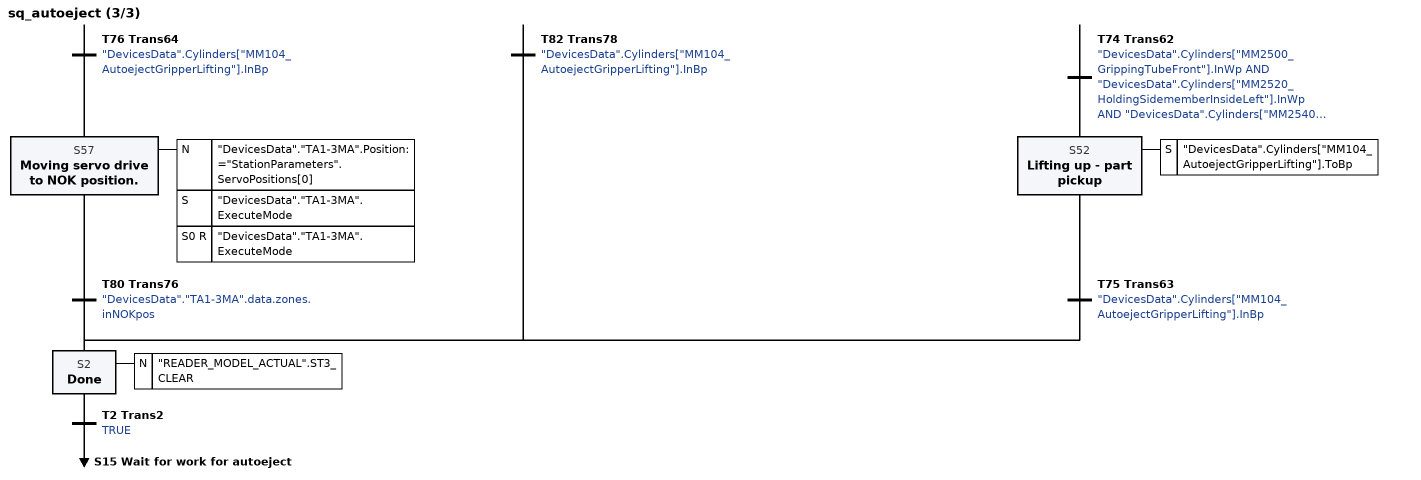
   // sequencer 1
   INITIAL_STEP Init:   // S1, max time T#10S, warning time T#7S
   END_STEP
   TRANSITION Trans1 FROM Init TO "Checking gripper status"   // T1
      := ("ModeSelection_DB".mode.activeMode = "mode_2_base") OR (("ModeSelection_DB".mode.activeMode = "mode_4_semiautomat") AND #start);
   END_TRANSITION
   STEP Done:   // S2, max time T#10S, warning time T#7S
              N    "READER_MODEL_ACTUAL".ST3_CLEAR
   END_STEP
   TRANSITION Trans2 FROM Done TO "Wait for work for autoeject"   // T2, jump
      := TRUE;
   END_TRANSITION
   STEP "Base done":   // S12, max time T#10S, warning time T#7S
   END_STEP
   TRANSITION Trans17 FROM "Base done" TO "Wait for work for autoeject"   // T17
      := (("ModeSelection_DB".mode.activeMode = "mode_3_automat") OR (("ModeSelection_DB".mode.activeMode = "mode_4_semiautomat") AND #start)) AND (#"Base done".T > t#2000MS);
   END_TRANSITION
   STEP "Wait for work for autoeject":   // S15, max time T#10S, warning time T#7S
   END_STEP
   TRANSITION "OK dropoff" FROM "Wait for work for autoeject" TO "Moving servo drive to OK position"   // T22
      := (("ModeSelection_DB".mode.activeMode = "mode_3_automat") OR (("ModeSelection_DB".mode.activeMode = "mode_4_semiautomat") AND #start)) AND "iR1outOf_AE_left_bottom" AND "iR1outOf_AE_left_top" AND "iR1outOf_AE_right_bottom" AND "iR1outOf_AE_right_top" AND "AutoPositions".AE_Gripper.PartPresent AND "AutoPositions".AE_Gripper.StFinished[3] AND NOT "AutoPositions".AE_Gripper.PartNOK AND "iAEtubePresentFront" AND "iAEtubePresentRear" AND NOT "AutoPositions".St4_OKposition.PartPresent AND NOT "i4partPresent";
   END_TRANSITION
   TRANSITION "NOK dropoff" FROM "Wait for work for autoeject" TO "Moving servo drive to NOK position.."   // T23
      := (("ModeSelection_DB".mode.activeMode = "mode_3_automat") OR (("ModeSelection_DB".mode.activeMode = "mode_4_semiautomat") AND #start)) AND "iR1outOf_AE_left_bottom" AND "iR1outOf_AE_left_top" AND "iR1outOf_AE_right_bottom" AND "iR1outOf_AE_right_top" AND "AutoPositions".AE_Gripper.PartPresent AND (NOT "AutoPositions".AE_Gripper.StFinished[3] OR "AutoPositions".AE_Gripper.PartNOK) AND "iAEtubePresentFront" AND "iAEtubePresentRear" AND NOT "PartHolderData".NOKBoxFull;
   END_TRANSITION
   TRANSITION "jig pickup" FROM "Wait for work for autoeject" TO "Moving servo drive to jig (st3) position"   // T21
      := (("ModeSelection_DB".mode.activeMode = "mode_3_automat") OR (("ModeSelection_DB".mode.activeMode = "mode_4_semiautomat") AND #start)) AND "iR1outOf_AE_left_bottom" AND "iR1outOf_AE_left_top" AND "iR1outOf_AE_right_bottom" AND "iR1outOf_AE_right_top" AND "AutoPositions".St3_Fitting.PartPresent AND "i3partPresent" AND NOT "AutoPositions".AE_Gripper.PartPresent AND NOT "iAEtubePresentFront" AND NOT "iAEtubePresentRear" AND NOT "AutoPositions".St4_OKposition.PartPresent AND NOT "i4partPresent";
   END_TRANSITION
   STEP "Close gripper - part pickup":   // S51, max time T#10S, warning time T#7S
              S    "DevicesData".Cylinders["MM2500_GrippingTubeFront"].ToWp
              S    "DevicesData".Cylinders["MM2520_HoldingSidememberInsideLeft"].ToWp
              S    "DevicesData".Cylinders["MM2540_HoldingSidememberOutsideLeft"].ToWp
   END_STEP
   TRANSITION Trans62 FROM "Close gripper - part pickup" TO "Lifting up - part pickup"   // T74
      := "DevicesData".Cylinders["MM2500_GrippingTubeFront"].InWp AND "DevicesData".Cylinders["MM2520_HoldingSidememberInsideLeft"].InWp AND "DevicesData".Cylinders["MM2540_HoldingSidememberOutsideLeft"].InWp;
   END_TRANSITION
   STEP "Open gripper - OK part dropoff":   // S53, max time T#10S, warning time T#7S
              S    "DevicesData".Cylinders["MM2500_GrippingTubeFront"].ToBp
              S    "DevicesData".Cylinders["MM2520_HoldingSidememberInsideLeft"].ToBp
              S    "DevicesData".Cylinders["MM2540_HoldingSidememberOutsideLeft"].ToBp
   END_STEP
   TRANSITION Trans75 FROM "Open gripper - OK part dropoff" TO "Lifting up - OK part dropoff"   // T79
      := "DevicesData".Cylinders["MM2500_GrippingTubeFront"].InBp AND "DevicesData".Cylinders["MM2520_HoldingSidememberInsideLeft"].InBp AND "DevicesData".Cylinders["MM2540_HoldingSidememberOutsideLeft"].InBp;
   END_TRANSITION
   STEP "Moving servo drive to OK position":   // S54, max time T#30S, warning time T#7S
      supervision V := #"Moving servo drive to OK position".T > #"Moving servo drive to OK position".T_MAX;
              N    "DevicesData"."TA1-3MA".Position:="StationParameters".ServoPositions[1]
              S    "DevicesData"."TA1-3MA".ExecuteMode
          S0  R    "DevicesData"."TA1-3MA".ExecuteMode
   END_STEP
   TRANSITION Trans74 FROM "Moving servo drive to OK position" TO "Lifting down - OK part dropoff"   // T78
      := "DevicesData"."TA1-3MA".data.zones.inOKpos;
   END_TRANSITION
   STEP "Lifting up - OK part dropoff":   // S55, max time T#10S, warning time T#7S
              S    "DevicesData".Cylinders["MM104_AutoejectGripperLifting"].ToBp
   END_STEP
   TRANSITION Trans64 FROM "Lifting up - OK part dropoff" TO "Moving servo drive to NOK position."   // T76
      := "DevicesData".Cylinders["MM104_AutoejectGripperLifting"].InBp;
   END_TRANSITION
   STEP "Lifting down - OK part dropoff":   // S56, max time T#10S, warning time T#7S
              S    "DevicesData".Cylinders["MM104_AutoejectGripperLifting"].ToWp
   END_STEP
   TRANSITION Trans73 FROM "Lifting down - OK part dropoff" TO "Open gripper - OK part dropoff"   // T77
      := "DevicesData".Cylinders["MM104_AutoejectGripperLifting"].InWp;
   END_TRANSITION
   STEP "Moving servo drive to jig (st3) position":   // S49, max time T#30S, warning time T#7S
      supervision V := #"Moving servo drive to jig (st3) position".T > #"Moving servo drive to jig (st3) position".T_MAX;
              N    "DevicesData"."TA1-3MA".Position:="StationParameters".ServoPositions[2]
              S    "DevicesData"."TA1-3MA".ExecuteMode
          S0  R    "DevicesData"."TA1-3MA".ExecuteMode
   END_STEP
   TRANSITION Trans85 FROM "Moving servo drive to jig (st3) position" TO "Waiting for part to be finished"   // T85
      := "DevicesData"."TA1-3MA".data.zones.inST3jig;
   END_TRANSITION
   STEP "Lifting up - part pickup":   // S52, max time T#10S, warning time T#7S
              S    "DevicesData".Cylinders["MM104_AutoejectGripperLifting"].ToBp
   END_STEP
   TRANSITION Trans63 FROM "Lifting up - part pickup" TO Done   // T75
      := "DevicesData".Cylinders["MM104_AutoejectGripperLifting"].InBp;
   END_TRANSITION
   STEP "Lifting down - part pickup":   // S50, max time T#10S, warning time T#7S
              S    "DevicesData".Cylinders["MM104_AutoejectGripperLifting"].ToWp
   END_STEP
   TRANSITION Trans61 FROM "Lifting down - part pickup" TO "Close gripper - part pickup"   // T73
      := "DevicesData".Cylinders["MM104_AutoejectGripperLifting"].InWp;
   END_TRANSITION
   STEP "Checking gripper status":   // S37, max time T#10S, warning time T#7S
   END_STEP
   TRANSITION "base w/o part" FROM "Checking gripper status" TO "Open gripper"   // T56
      := NOT "AutoPositions".AE_Gripper.PartPresent AND NOT "iAEtubePresentFront" AND NOT "iAEtubePresentRear";
   END_TRANSITION
   TRANSITION "base w/ part" FROM "Checking gripper status" TO "Close gripper"   // T57
      := "AutoPositions".AE_Gripper.PartPresent AND "iAEtubePresentFront" AND "iAEtubePresentRear";
   END_TRANSITION
   STEP "Open gripper":   // S38, max time T#10S, warning time T#7S
              S    "DevicesData".Cylinders["MM2500_GrippingTubeFront"].ToBp
              S    "DevicesData".Cylinders["MM2520_HoldingSidememberInsideLeft"].ToBp
              S    "DevicesData".Cylinders["MM2540_HoldingSidememberOutsideLeft"].ToBp
   END_STEP
   TRANSITION Trans58 FROM "Open gripper" TO "Lifting up"   // T58
      := "DevicesData".Cylinders["MM2500_GrippingTubeFront"].InBp AND "DevicesData".Cylinders["MM2520_HoldingSidememberInsideLeft"].InBp AND "DevicesData".Cylinders["MM2540_HoldingSidememberOutsideLeft"].InBp;
   END_TRANSITION
   STEP "Close gripper":   // S39, max time T#10S, warning time T#7S
              S    "DevicesData".Cylinders["MM2500_GrippingTubeFront"].ToWp
              S    "DevicesData".Cylinders["MM2520_HoldingSidememberInsideLeft"].ToWp
              S    "DevicesData".Cylinders["MM2540_HoldingSidememberOutsideLeft"].ToWp
   END_STEP
   TRANSITION Trans59 FROM "Close gripper" TO "Lifting up"   // T59
      := "DevicesData".Cylinders["MM2500_GrippingTubeFront"].InWp AND "DevicesData".Cylinders["MM2520_HoldingSidememberInsideLeft"].InWp AND "DevicesData".Cylinders["MM2540_HoldingSidememberOutsideLeft"].InWp;
   END_TRANSITION
   STEP "Lifting up":   // S40, max time T#10S, warning time T#7S
              S    "DevicesData".Cylinders["MM104_AutoejectGripperLifting"].ToBp
   END_STEP
   TRANSITION Trans60 FROM "Lifting up" TO "Checking homing status"   // T60
      := "DevicesData".Cylinders["MM104_AutoejectGripperLifting"].InBp;
   END_TRANSITION
   STEP "Checking homing status":   // S41, max time T#10S, warning time T#7S
   END_STEP
   TRANSITION referenced FROM "Checking homing status" TO "Checking robot position."   // T61
      := "DevicesData"."TA1-3MA".AxisRef;
   END_TRANSITION
   TRANSITION "not refrenced" FROM "Checking homing status" TO "Checking robot position"   // T62
      := NOT "DevicesData"."TA1-3MA".AxisRef;
   END_TRANSITION
   STEP "Checking robot position":   // S42, max time T#10S, warning time T#7S
   END_STEP
   TRANSITION "out of zones" FROM "Checking robot position" TO "Switch servo to homing mode"   // T63
      := "iR1outOf_AE_left_bottom" AND "iR1outOf_AE_left_top" AND "iR1outOf_AE_right_bottom" AND "iR1outOf_AE_right_top";
   END_TRANSITION
   TRANSITION "in zones" FROM "Checking robot position" TO "You have to move robot out of the autoeject zones manually"   // T64
      := TRUE;
   END_TRANSITION
   STEP "Switch servo to homing mode":   // S43, max time T#10S, warning time T#7S
      supervision V := #"Switch servo to homing mode".T > #"Switch servo to homing mode".T_MAX;
              N    "DevicesData"."TA1-3MA".ModePos:=4
   END_STEP
   TRANSITION Trans65 FROM "Switch servo to homing mode" TO "Homing servo drive"   // T65
      := "DevicesData"."TA1-3MA".ActMode = 4;
   END_TRANSITION
   STEP "You have to move robot out of the autoeject zones manually":   // S44, max time T#10S, warning time T#7S
      supervision V := "AlwaysTRUE";
   END_STEP
   TRANSITION Trans66 FROM "You have to move robot out of the autoeject zones manually" TO END   // T66
      := NOT "AlwaysTRUE";
   END_TRANSITION
   STEP "Homing servo drive":   // S45, max time T#30S, warning time T#7S
      supervision V := #"Homing servo drive".T > #"Homing servo drive".T_MAX;
              S    "DevicesData"."TA1-3MA".ExecuteMode
          S0  R    "DevicesData"."TA1-3MA".ExecuteMode
   END_STEP
   TRANSITION Trans67 FROM "Homing servo drive" TO "Checking robot position."   // T67
      := "DevicesData"."TA1-3MA".AxisRef AND "DevicesData"."TA1-3MA".AxisPosOk;
   END_TRANSITION
   STEP "Checking robot position.":   // S46, max time T#10S, warning time T#7S
   END_STEP
   TRANSITION Trans68 FROM "Checking robot position." TO "Switch servo to positioning mode"   // T68
      := ("iR1outOf_AE_left_bottom" AND "iR1outOf_AE_left_top" AND "iR1outOf_AE_right_bottom" AND "iR1outOf_AE_right_top") OR ("iR1outOf_AE_right_bottom" AND "iR1outOf_AE_right_top" AND "DevicesData"."TA1-3MA".data.zones.outOfST3zone);
   END_TRANSITION
   TRANSITION Trans69 FROM "Checking robot position." TO "You have to move robot out of the autoeject zones manually"   // T69, jump
      := TRUE;
   END_TRANSITION
   STEP "Switch servo to positioning mode":   // S47, max time T#10S, warning time T#7S
      supervision V := #"Switch servo to positioning mode".T > #"Switch servo to positioning mode".T_MAX;
              N    "DevicesData"."TA1-3MA".ModePos:=2
   END_STEP
   TRANSITION Trans70 FROM "Switch servo to positioning mode" TO Timeout   // T70
      := "DevicesData"."TA1-3MA".ActMode = 2;
   END_TRANSITION
   STEP "Moving servo drive to NOK position":   // S48, max time T#30S, warning time T#7S
      supervision V := #"Moving servo drive to NOK position".T > #"Moving servo drive to NOK position".T_MAX;
              N    "DevicesData"."TA1-3MA".Position:="StationParameters".ServoPositions[0]
              S    "DevicesData"."TA1-3MA".ExecuteMode
          S0  R    "DevicesData"."TA1-3MA".ExecuteMode
   END_STEP
   TRANSITION Trans71 FROM "Moving servo drive to NOK position" TO "Base done"   // T71
      := "DevicesData"."TA1-3MA".data.zones.inNOKpos;
   END_TRANSITION
   STEP "Moving servo drive to NOK position.":   // S57, max time T#30S, warning time T#7S
      supervision V := #"Moving servo drive to NOK position.".T > #"Moving servo drive to NOK position.".T_MAX;
              N    "DevicesData"."TA1-3MA".Position:="StationParameters".ServoPositions[0]
              S    "DevicesData"."TA1-3MA".ExecuteMode
          S0  R    "DevicesData"."TA1-3MA".ExecuteMode
   END_STEP
   TRANSITION Trans76 FROM "Moving servo drive to NOK position." TO Done   // T80
      := "DevicesData"."TA1-3MA".data.zones.inNOKpos;
   END_TRANSITION
   STEP "Open gripper - NOK part dropoff":   // S58, max time T#10S, warning time T#7S
              S    "DevicesData".Cylinders["MM2500_GrippingTubeFront"].ToBp
              S    "DevicesData".Cylinders["MM2520_HoldingSidememberInsideLeft"].ToBp
              S    "DevicesData".Cylinders["MM2540_HoldingSidememberOutsideLeft"].ToBp
   END_STEP
   TRANSITION Trans80 FROM "Open gripper - NOK part dropoff" TO "Lifting up - NOK part dropoff"   // T84
      := "DevicesData".Cylinders["MM2500_GrippingTubeFront"].InBp AND "DevicesData".Cylinders["MM2520_HoldingSidememberInsideLeft"].InBp AND "DevicesData".Cylinders["MM2540_HoldingSidememberOutsideLeft"].InBp;
   END_TRANSITION
   STEP "Moving servo drive to NOK position..":   // S59, max time T#30S, warning time T#7S
      supervision V := #"Moving servo drive to NOK position..".T > #"Moving servo drive to NOK position..".T_MAX;
              N    "DevicesData"."TA1-3MA".Position:="StationParameters".ServoPositions[0]
              S    "DevicesData"."TA1-3MA".ExecuteMode
          S0  R    "DevicesData"."TA1-3MA".ExecuteMode
   END_STEP
   TRANSITION Trans79 FROM "Moving servo drive to NOK position.." TO "Lifting down - NOK part dropoff"   // T83
      := "DevicesData"."TA1-3MA".data.zones.inNOKpos;
   END_TRANSITION
   STEP "Lifting up - NOK part dropoff":   // S60, max time T#10S, warning time T#7S
              S    "DevicesData".Cylinders["MM104_AutoejectGripperLifting"].ToBp
   END_STEP
   TRANSITION Trans78 FROM "Lifting up - NOK part dropoff" TO Done   // T82
      := "DevicesData".Cylinders["MM104_AutoejectGripperLifting"].InBp;
   END_TRANSITION
   STEP "Lifting down - NOK part dropoff":   // S61, max time T#10S, warning time T#7S
              S    "DevicesData".Cylinders["MM104_AutoejectGripperLifting"].ToWp
   END_STEP
   TRANSITION Trans77 FROM "Lifting down - NOK part dropoff" TO "Open gripper - NOK part dropoff"   // T81
      := "DevicesData".Cylinders["MM104_AutoejectGripperLifting"].InWp;
   END_TRANSITION
   STEP "Waiting for part to be finished":   // S62, max time T#10S, warning time T#7S
   END_STEP
   TRANSITION Trans72 FROM "Waiting for part to be finished" TO "Lifting down - part pickup"   // T72
      := "sq_fitting_station_st3"."Ready for pickup by autoeject".X AND "sq_fitting_station_st3".base AND "AutoPositions".St3_Fitting.PartPresent AND "i3partPresent" AND NOT "AutoPositions".AE_Gripper.PartPresent AND NOT "iAEtubePresentFront" AND NOT "iAEtubePresentRear" AND NOT "AutoPositions".St4_OKposition.PartPresent;
   END_TRANSITION
   STEP Timeout:   // S63, max time T#10S, warning time T#7S
   END_STEP
   TRANSITION Trans86 FROM Timeout TO "Moving servo drive to NOK position"   // T86
      := #Timeout.T > t#100MS;
   END_TRANSITION
END_FUNCTION_BLOCK

FUNCTION_BLOCK "sq_carousel_main"   // FB70, GRAPH
VERSION : 0.1
// stored: AcknowledgeErrorsRequired true, AutoNumber true, GraphVersion 6.0, InitialValuesAcquisition false, IsIECCheckEnabled false, LanguageInNetworks LAD, LockOperatingMode false, PermanentILProcessingInMANMode false, SetENOAutomatically false, SkipSteps false, UDAEnableTagReadback false, WithAlarmHandling true
   // inherited from GRAPH_BASE
   VAR
      OFF_SQ_BASE : Bool;
   END_VAR
   VAR_INPUT
      OFF_SQ { ExternalAccessible := 'False'; ExternalVisible := 'False'; ExternalWritable := 'False'} : Bool := false;   // Turn sequence off
      INIT_SQ { ExternalAccessible := 'False'; ExternalVisible := 'False'; ExternalWritable := 'False'} : Bool := false;   // Set sequence to initial state
      ACK_EF { ExternalAccessible := 'False'; ExternalVisible := 'False'; ExternalWritable := 'False'} : Bool := false;   // Acknowledge all errors and faults
      S_PREV { ExternalAccessible := 'False'; ExternalVisible := 'False'; ExternalWritable := 'False'} : Bool := false;   // Output previous step in parameter S_NO
      S_NEXT { ExternalAccessible := 'False'; ExternalVisible := 'False'; ExternalWritable := 'False'} : Bool := false;   // Indicate next step in parameter S_NO
      SW_AUTO { ExternalAccessible := 'False'; ExternalVisible := 'False'; ExternalWritable := 'False'} : Bool := false;   // Automatic mode
      SW_TAP { ExternalAccessible := 'False'; ExternalVisible := 'False'; ExternalWritable := 'False'} : Bool := false;   // Semiautomatic/switch with transition
      SW_TOP { ExternalAccessible := 'False'; ExternalVisible := 'False'; ExternalWritable := 'False'} : Bool := false;   // Semiautomatic/ignore transition
      SW_MAN { ExternalAccessible := 'False'; ExternalVisible := 'False'; ExternalWritable := 'False'} : Bool := false;   // Manual mode
      S_SEL { ExternalAccessible := 'False'; ExternalVisible := 'False'; ExternalWritable := 'False'} : Int := 0;   // Select step to be output to S_NO
      S_ON { ExternalAccessible := 'False'; ExternalVisible := 'False'; ExternalWritable := 'False'} : Bool := false;   // Activate step indicated in S_NO
      S_OFF { ExternalAccessible := 'False'; ExternalVisible := 'False'; ExternalWritable := 'False'} : Bool := false;   // Deactivate step indicated S_NO
      T_PUSH { ExternalAccessible := 'False'; ExternalVisible := 'False'; ExternalWritable := 'False'} : Bool := false;   // Enable transition to switch in semi automatic mode
   END_VAR
   VAR_OUTPUT
      S_NO { ExternalAccessible := 'False'; ExternalVisible := 'False'; ExternalWritable := 'False'} : Int := 0;   // Step number
      S_MORE { ExternalAccessible := 'False'; ExternalVisible := 'False'; ExternalWritable := 'False'} : Bool := false;   // More steps are available and can be shown in S_NO
      S_ACTIVE { ExternalAccessible := 'False'; ExternalVisible := 'False'; ExternalWritable := 'False'} : Bool := false;   // Step indicated in S_NO is active
      ERR_FLT { ExternalAccessible := 'False'; ExternalVisible := 'False'; ExternalWritable := 'False'} : Bool := false;   // Interlock or supervision group error
      AUTO_ON { ExternalAccessible := 'False'; ExternalVisible := 'False'; ExternalWritable := 'False'} : Bool := false;   // Automatic mode is active
      TAP_ON { ExternalAccessible := 'False'; ExternalVisible := 'False'; ExternalWritable := 'False'} : Bool := false;   // Semiautomatic mode/step with transition enabled
      TOP_ON { ExternalAccessible := 'False'; ExternalVisible := 'False'; ExternalWritable := 'False'} : Bool := false;   // Semiautomatic mode/ignore transition enabled
      MAN_ON { ExternalAccessible := 'False'; ExternalVisible := 'False'; ExternalWritable := 'False'} : Bool := false;   // Manual mode is active
   END_VAR
   VAR
      dummy : Bool;
      start : Bool;
      base : Bool;
   END_VAR
BEGIN
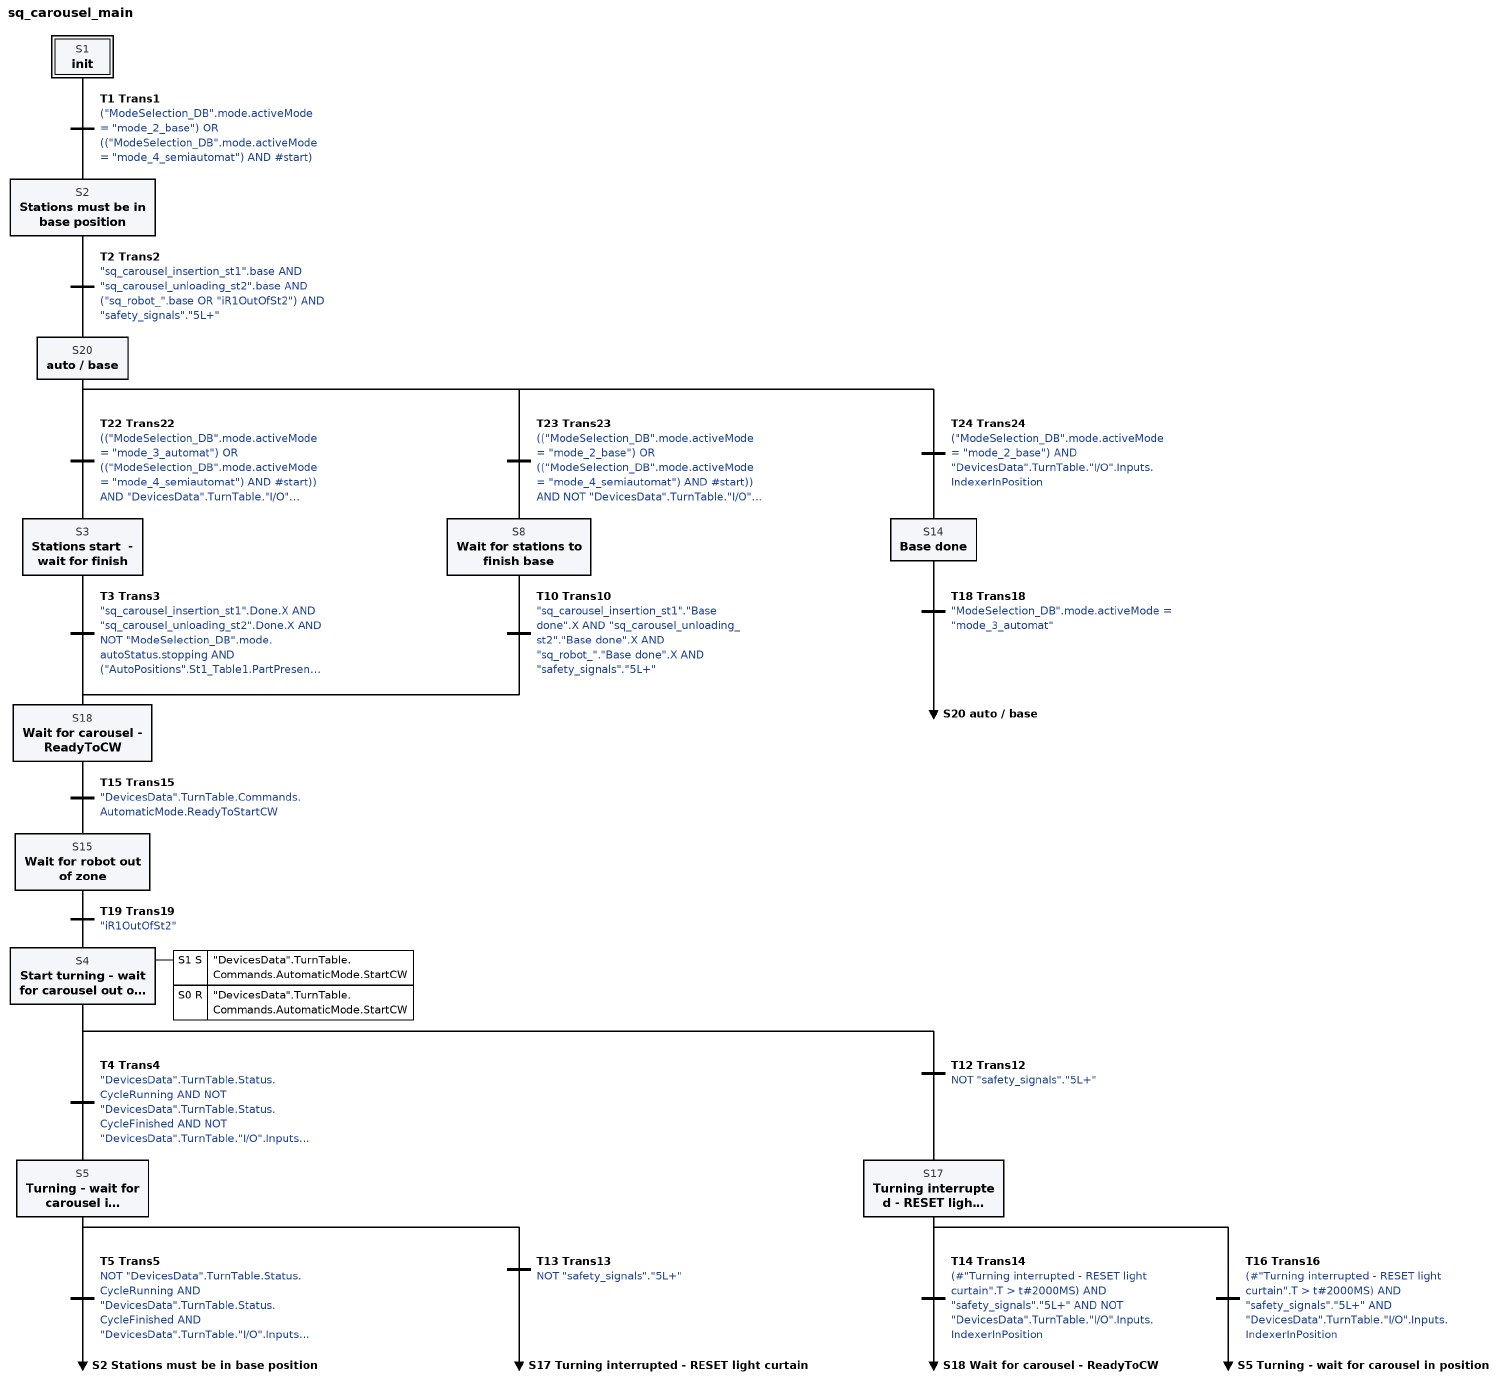
   // permanent pre-instructions
   NETWORK 1
      #base := "iTurnTableIndexerInPosition";

   // sequencer 1
   INITIAL_STEP init:   // S1, max time T#10S, warning time T#7S
   END_STEP
   TRANSITION Trans1 FROM init TO "Stations must be in base position"   // T1
      := ("ModeSelection_DB".mode.activeMode = "mode_2_base") OR (("ModeSelection_DB".mode.activeMode = "mode_4_semiautomat") AND #start);
   END_TRANSITION
   STEP "Stations must be in base position":   // S2, max time T#10S, warning time T#7S
      supervision V := #"Stations must be in base position".T > #"Stations must be in base position".T_MAX;
   END_STEP
   TRANSITION Trans2 FROM "Stations must be in base position" TO "auto / base"   // T2
      := "sq_carousel_insertion_st1".base AND "sq_carousel_unloading_st2".base AND ("sq_robot_".base OR "iR1OutOfSt2") AND "safety_signals"."5L+";
   END_TRANSITION
   STEP "Stations start  - wait for finish":   // S3, max time T#10S, warning time T#7S
   END_STEP
   TRANSITION Trans3 FROM "Stations start  - wait for finish" TO "Wait for carousel - ReadyToCW"   // T3
      := "sq_carousel_insertion_st1".Done.X AND "sq_carousel_unloading_st2".Done.X AND NOT "ModeSelection_DB".mode.autoStatus.stopping AND ("AutoPositions".St1_Table1.PartPresent OR "AutoPositions".St2_Table2.PartPresent OR NOT "ModeSelection_DB".mode.autoStatus.emptying) AND "safety_signals"."5L+";
   END_TRANSITION
   STEP "Start turning - wait for carousel out of position":   // S4, max time T#10S, warning time T#7S
      supervision V := #"Start turning - wait for carousel out of position".T > #"Start turning - wait for carousel out of position".T_MAX;
          S1  S    "DevicesData".TurnTable.Commands.AutomaticMode.StartCW
          S0  R    "DevicesData".TurnTable.Commands.AutomaticMode.StartCW
   END_STEP
   TRANSITION Trans4 FROM "Start turning - wait for carousel out of position" TO "Turning - wait for carousel in position"   // T4
      := "DevicesData".TurnTable.Status.CycleRunning AND NOT "DevicesData".TurnTable.Status.CycleFinished AND NOT "DevicesData".TurnTable."I/O".Inputs.IndexerInPosition;
   END_TRANSITION
   TRANSITION Trans12 FROM "Start turning - wait for carousel out of position" TO "Turning interrupted - RESET light curtain"   // T12
      := NOT "safety_signals"."5L+";
   END_TRANSITION
   STEP "Turning - wait for carousel in position":   // S5, max time T#10S, warning time T#7S
      supervision V := #"Turning - wait for carousel in position".T > #"Turning - wait for carousel in position".T_MAX;
   END_STEP
   TRANSITION Trans5 FROM "Turning - wait for carousel in position" TO "Stations must be in base position"   // T5, jump
      := NOT "DevicesData".TurnTable.Status.CycleRunning AND "DevicesData".TurnTable.Status.CycleFinished AND "DevicesData".TurnTable."I/O".Inputs.IndexerInPosition;
   END_TRANSITION
   TRANSITION Trans13 FROM "Turning - wait for carousel in position" TO "Turning interrupted - RESET light curtain"   // T13, jump
      := NOT "safety_signals"."5L+";
   END_TRANSITION
   STEP "Turning interrupted - RESET light curtain":   // S17, max time T#10S, warning time T#7S
   END_STEP
   TRANSITION Trans14 FROM "Turning interrupted - RESET light curtain" TO "Wait for carousel - ReadyToCW"   // T14, jump
      := (#"Turning interrupted - RESET light curtain".T > t#2000MS) AND "safety_signals"."5L+" AND NOT "DevicesData".TurnTable."I/O".Inputs.IndexerInPosition;
   END_TRANSITION
   TRANSITION Trans16 FROM "Turning interrupted - RESET light curtain" TO "Turning - wait for carousel in position"   // T16, jump
      := (#"Turning interrupted - RESET light curtain".T > t#2000MS) AND "safety_signals"."5L+" AND "DevicesData".TurnTable."I/O".Inputs.IndexerInPosition;
   END_TRANSITION
   STEP "Wait for carousel - ReadyToCW":   // S18, max time T#10S, warning time T#7S
      supervision V := #"Wait for carousel - ReadyToCW".T > #"Wait for carousel - ReadyToCW".T_MAX;
   END_STEP
   TRANSITION Trans15 FROM "Wait for carousel - ReadyToCW" TO "Wait for robot out of zone"   // T15
      := "DevicesData".TurnTable.Commands.AutomaticMode.ReadyToStartCW;
   END_TRANSITION
   STEP "Wait for stations to finish base":   // S8, max time T#10S, warning time T#7S
   END_STEP
   TRANSITION Trans10 FROM "Wait for stations to finish base" TO "Wait for carousel - ReadyToCW"   // T10
      := "sq_carousel_insertion_st1"."Base done".X AND "sq_carousel_unloading_st2"."Base done".X AND "sq_robot_"."Base done".X AND "safety_signals"."5L+";
   END_TRANSITION
   STEP "auto / base":   // S20, max time T#10S, warning time T#7S
   END_STEP
   TRANSITION Trans22 FROM "auto / base" TO "Stations start  - wait for finish"   // T22
      := (("ModeSelection_DB".mode.activeMode = "mode_3_automat") OR (("ModeSelection_DB".mode.activeMode = "mode_4_semiautomat") AND #start)) AND "DevicesData".TurnTable."I/O".Inputs.IndexerInPosition;
   END_TRANSITION
   TRANSITION Trans23 FROM "auto / base" TO "Wait for stations to finish base"   // T23
      := (("ModeSelection_DB".mode.activeMode = "mode_2_base") OR (("ModeSelection_DB".mode.activeMode = "mode_4_semiautomat") AND #start)) AND NOT "DevicesData".TurnTable."I/O".Inputs.IndexerInPosition;
   END_TRANSITION
   TRANSITION Trans24 FROM "auto / base" TO "Base done"   // T24
      := ("ModeSelection_DB".mode.activeMode = "mode_2_base") AND "DevicesData".TurnTable."I/O".Inputs.IndexerInPosition;
   END_TRANSITION
   STEP "Base done":   // S14, max time T#10S, warning time T#7S
   END_STEP
   TRANSITION Trans18 FROM "Base done" TO "auto / base"   // T18, jump
      := "ModeSelection_DB".mode.activeMode = "mode_3_automat";
   END_TRANSITION
   STEP "Wait for robot out of zone":   // S15, max time T#10S, warning time T#7S
      supervision V := #"Wait for robot out of zone".T > #"Wait for robot out of zone".T_MAX;
   END_STEP
   TRANSITION Trans19 FROM "Wait for robot out of zone" TO "Start turning - wait for carousel out of position"   // T19
      := "iR1OutOfSt2";
   END_TRANSITION
END_FUNCTION_BLOCK

FUNCTION_BLOCK "sq_carousel_st1"   // FB39, GRAPH
VERSION : 0.1
// stored: AcknowledgeErrorsRequired true, AutoNumber true, GraphVersion 6.0, InitialValuesAcquisition false, IsIECCheckEnabled false, LanguageInNetworks LAD, LockOperatingMode false, PermanentILProcessingInMANMode false, SetENOAutomatically false, SkipSteps false, UDAEnableTagReadback false, WithAlarmHandling true
   // inherited from GRAPH_BASE
   VAR
      OFF_SQ_BASE : Bool;
   END_VAR
   VAR_INPUT
      OFF_SQ { ExternalAccessible := 'False'; ExternalVisible := 'False'; ExternalWritable := 'False'} : Bool := false;   // Turn sequence off
      INIT_SQ { ExternalAccessible := 'False'; ExternalVisible := 'False'; ExternalWritable := 'False'} : Bool := false;   // Set sequence to initial state
      ACK_EF { ExternalAccessible := 'False'; ExternalVisible := 'False'; ExternalWritable := 'False'} : Bool := false;   // Acknowledge all errors and faults
      S_PREV { ExternalAccessible := 'False'; ExternalVisible := 'False'; ExternalWritable := 'False'} : Bool := false;   // Output previous step in parameter S_NO
      S_NEXT { ExternalAccessible := 'False'; ExternalVisible := 'False'; ExternalWritable := 'False'} : Bool := false;   // Indicate next step in parameter S_NO
      SW_AUTO { ExternalAccessible := 'False'; ExternalVisible := 'False'; ExternalWritable := 'False'} : Bool := false;   // Automatic mode
      SW_TAP { ExternalAccessible := 'False'; ExternalVisible := 'False'; ExternalWritable := 'False'} : Bool := false;   // Semiautomatic/switch with transition
      SW_TOP { ExternalAccessible := 'False'; ExternalVisible := 'False'; ExternalWritable := 'False'} : Bool := false;   // Semiautomatic/ignore transition
      SW_MAN { ExternalAccessible := 'False'; ExternalVisible := 'False'; ExternalWritable := 'False'} : Bool := false;   // Manual mode
      S_SEL { ExternalAccessible := 'False'; ExternalVisible := 'False'; ExternalWritable := 'False'} : Int := 0;   // Select step to be output to S_NO
      S_ON { ExternalAccessible := 'False'; ExternalVisible := 'False'; ExternalWritable := 'False'} : Bool := false;   // Activate step indicated in S_NO
      S_OFF { ExternalAccessible := 'False'; ExternalVisible := 'False'; ExternalWritable := 'False'} : Bool := false;   // Deactivate step indicated S_NO
      T_PUSH { ExternalAccessible := 'False'; ExternalVisible := 'False'; ExternalWritable := 'False'} : Bool := false;   // Enable transition to switch in semi automatic mode
   END_VAR
   VAR_OUTPUT
      S_NO { ExternalAccessible := 'False'; ExternalVisible := 'False'; ExternalWritable := 'False'} : Int := 0;   // Step number
      S_MORE { ExternalAccessible := 'False'; ExternalVisible := 'False'; ExternalWritable := 'False'} : Bool := false;   // More steps are available and can be shown in S_NO
      S_ACTIVE { ExternalAccessible := 'False'; ExternalVisible := 'False'; ExternalWritable := 'False'} : Bool := false;   // Step indicated in S_NO is active
      ERR_FLT { ExternalAccessible := 'False'; ExternalVisible := 'False'; ExternalWritable := 'False'} : Bool := false;   // Interlock or supervision group error
      AUTO_ON { ExternalAccessible := 'False'; ExternalVisible := 'False'; ExternalWritable := 'False'} : Bool := false;   // Automatic mode is active
      TAP_ON { ExternalAccessible := 'False'; ExternalVisible := 'False'; ExternalWritable := 'False'} : Bool := false;   // Semiautomatic mode/step with transition enabled
      TOP_ON { ExternalAccessible := 'False'; ExternalVisible := 'False'; ExternalWritable := 'False'} : Bool := false;   // Semiautomatic mode/ignore transition enabled
      MAN_ON { ExternalAccessible := 'False'; ExternalVisible := 'False'; ExternalWritable := 'False'} : Bool := false;   // Manual mode is active
   END_VAR
   VAR
      dummy : Bool;
      start : Bool;
      base : Bool;
      startEmpty : Bool;
   END_VAR
   VAR_TEMP   // added for the SCL form of the ladder/FBD networks
      _w1 : Bool;
      _w2 : Bool;
   END_VAR
BEGIN
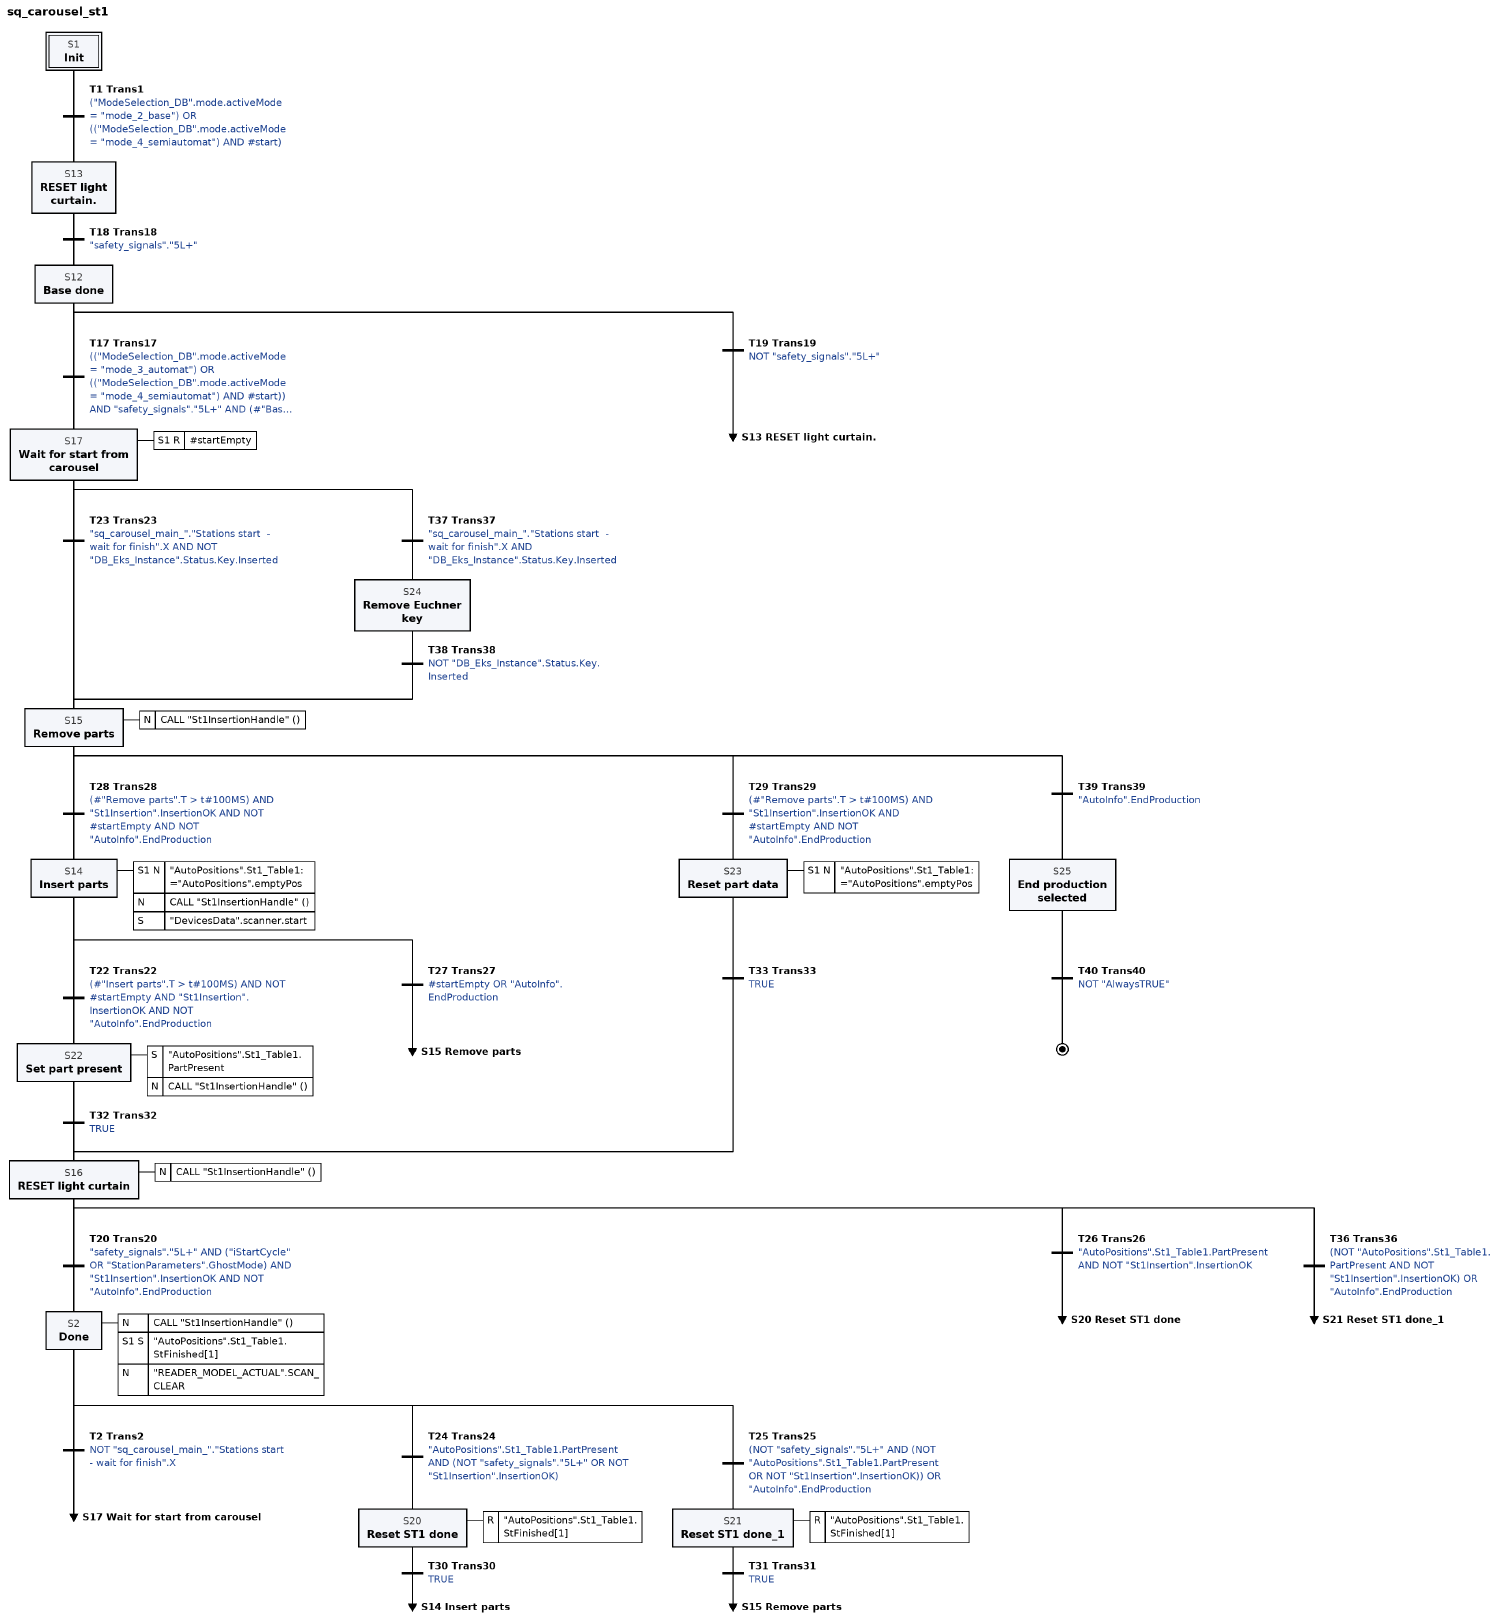
   // permanent pre-instructions
   NETWORK 1
      #base := TRUE;
   NETWORK 2
      "St1Insertion".ExpectedSensors := "St1Insertion".EmptyBits;
      #_w1 := ("ModeSelection_DB".mode.activeMode = "mode_3_automat") OR ("ModeSelection_DB".mode.activeMode = "mode_4_semiautomat");
      IF #_w1 THEN "St1Insertion".UsedSensors := "St1Insertion".FullBits; END_IF;
      IF NOT #_w1 THEN "St1Insertion".UsedSensors := "St1Insertion".EmptyBits; END_IF;
      #_w2 := ("AutoPositions".St1_Table1.PartPresent OR #"Insert parts".X) AND NOT #startEmpty AND NOT "StationParameters".GhostMode AND NOT #"Remove parts".X;
      IF #_w2 THEN
          MOVE_BLK(IN := "DB_ProductionProgramActual".Program.St1Insertion[1],
                   COUNT := 20,
                   OUT => "St1Insertion".ExpectedSensors[1]);
          MOVE_BLK(IN := "DB_ProductionProgramActual".Program.St1InsertionUsed[1],
                   COUNT := 20,
                   OUT => "St1Insertion".UsedSensors[1]);
      END_IF;
      "St1InsertionHandle"();

   // sequencer 1
   INITIAL_STEP Init:   // S1, max time T#10S, warning time T#7S
   END_STEP
   TRANSITION Trans1 FROM Init TO "RESET light curtain."   // T1
      := ("ModeSelection_DB".mode.activeMode = "mode_2_base") OR (("ModeSelection_DB".mode.activeMode = "mode_4_semiautomat") AND #start);
   END_TRANSITION
   STEP Done:   // S2, max time T#10S, warning time T#7S
              N    CALL "St1InsertionHandle" ()
          S1  S    "AutoPositions".St1_Table1.StFinished[1]
              N    "READER_MODEL_ACTUAL".SCAN_CLEAR
   END_STEP
   TRANSITION Trans2 FROM Done TO "Wait for start from carousel"   // T2, jump
      := NOT "sq_carousel_main_"."Stations start  - wait for finish".X;
   END_TRANSITION
   TRANSITION Trans24 FROM Done TO "Reset ST1 done"   // T24
      := "AutoPositions".St1_Table1.PartPresent AND (NOT "safety_signals"."5L+" OR NOT "St1Insertion".InsertionOK);
   END_TRANSITION
   TRANSITION Trans25 FROM Done TO "Reset ST1 done_1"   // T25
      := (NOT "safety_signals"."5L+" AND (NOT "AutoPositions".St1_Table1.PartPresent OR NOT "St1Insertion".InsertionOK)) OR "AutoInfo".EndProduction;
   END_TRANSITION
   STEP "Base done":   // S12, max time T#10S, warning time T#7S
   END_STEP
   TRANSITION Trans17 FROM "Base done" TO "Wait for start from carousel"   // T17
      := (("ModeSelection_DB".mode.activeMode = "mode_3_automat") OR (("ModeSelection_DB".mode.activeMode = "mode_4_semiautomat") AND #start)) AND "safety_signals"."5L+" AND (#"Base done".T > t#2000MS);
   END_TRANSITION
   TRANSITION Trans19 FROM "Base done" TO "RESET light curtain."   // T19, jump
      := NOT "safety_signals"."5L+";
   END_TRANSITION
   STEP "RESET light curtain.":   // S13, max time T#10S, warning time T#7S
   END_STEP
   TRANSITION Trans18 FROM "RESET light curtain." TO "Base done"   // T18
      := "safety_signals"."5L+";
   END_TRANSITION
   STEP "Insert parts":   // S14, max time T#10S, warning time T#7S
          S1  N    "AutoPositions".St1_Table1:="AutoPositions".emptyPos
              N    CALL "St1InsertionHandle" ()
              S    "DevicesData".scanner.start
   END_STEP
   TRANSITION Trans22 FROM "Insert parts" TO "Set part present"   // T22
      := (#"Insert parts".T > t#100MS) AND NOT #startEmpty AND "St1Insertion".InsertionOK AND NOT "AutoInfo".EndProduction;
   END_TRANSITION
   TRANSITION Trans27 FROM "Insert parts" TO "Remove parts"   // T27, jump
      := #startEmpty OR "AutoInfo".EndProduction;
   END_TRANSITION
   STEP "Remove parts":   // S15, max time T#10S, warning time T#7S
              N    CALL "St1InsertionHandle" ()
   END_STEP
   TRANSITION Trans28 FROM "Remove parts" TO "Insert parts"   // T28
      := (#"Remove parts".T > t#100MS) AND "St1Insertion".InsertionOK AND NOT #startEmpty AND NOT "AutoInfo".EndProduction;
   END_TRANSITION
   TRANSITION Trans29 FROM "Remove parts" TO "Reset part data"   // T29
      := (#"Remove parts".T > t#100MS) AND "St1Insertion".InsertionOK AND #startEmpty AND NOT "AutoInfo".EndProduction;
   END_TRANSITION
   TRANSITION Trans39 FROM "Remove parts" TO "End production selected"   // T39
      := "AutoInfo".EndProduction;
   END_TRANSITION
   STEP "RESET light curtain":   // S16, max time T#10S, warning time T#7S
              N    CALL "St1InsertionHandle" ()
   END_STEP
   TRANSITION Trans20 FROM "RESET light curtain" TO Done   // T20
      := "safety_signals"."5L+" AND ("iStartCycle" OR "StationParameters".GhostMode) AND "St1Insertion".InsertionOK AND NOT "AutoInfo".EndProduction;
   END_TRANSITION
   TRANSITION Trans26 FROM "RESET light curtain" TO "Reset ST1 done"   // T26, jump
      := "AutoPositions".St1_Table1.PartPresent AND NOT "St1Insertion".InsertionOK;
   END_TRANSITION
   TRANSITION Trans36 FROM "RESET light curtain" TO "Reset ST1 done_1"   // T36, jump
      := (NOT "AutoPositions".St1_Table1.PartPresent AND NOT "St1Insertion".InsertionOK) OR "AutoInfo".EndProduction;
   END_TRANSITION
   STEP "Wait for start from carousel":   // S17, max time T#10S, warning time T#7S
          S1  R    #startEmpty
   END_STEP
   TRANSITION Trans23 FROM "Wait for start from carousel" TO "Remove parts"   // T23
      := "sq_carousel_main_"."Stations start  - wait for finish".X AND NOT "DB_Eks_Instance".Status.Key.Inserted;
   END_TRANSITION
   TRANSITION Trans37 FROM "Wait for start from carousel" TO "Remove Euchner key"   // T37
      := "sq_carousel_main_"."Stations start  - wait for finish".X AND "DB_Eks_Instance".Status.Key.Inserted;
   END_TRANSITION
   STEP "Reset ST1 done":   // S20, max time T#10S, warning time T#7S
              R    "AutoPositions".St1_Table1.StFinished[1]
   END_STEP
   TRANSITION Trans30 FROM "Reset ST1 done" TO "Insert parts"   // T30, jump
      := TRUE;
   END_TRANSITION
   STEP "Reset ST1 done_1":   // S21, max time T#10S, warning time T#7S
              R    "AutoPositions".St1_Table1.StFinished[1]
   END_STEP
   TRANSITION Trans31 FROM "Reset ST1 done_1" TO "Remove parts"   // T31, jump
      := TRUE;
   END_TRANSITION
   STEP "Set part present":   // S22, max time T#10S, warning time T#7S
              S    "AutoPositions".St1_Table1.PartPresent
              N    CALL "St1InsertionHandle" ()
   END_STEP
   TRANSITION Trans32 FROM "Set part present" TO "RESET light curtain"   // T32
      := TRUE;
   END_TRANSITION
   STEP "Reset part data":   // S23, max time T#10S, warning time T#7S
          S1  N    "AutoPositions".St1_Table1:="AutoPositions".emptyPos
   END_STEP
   TRANSITION Trans33 FROM "Reset part data" TO "RESET light curtain"   // T33
      := TRUE;
   END_TRANSITION
   STEP "Remove Euchner key":   // S24, max time T#10S, warning time T#7S
   END_STEP
   TRANSITION Trans38 FROM "Remove Euchner key" TO "Remove parts"   // T38
      := NOT "DB_Eks_Instance".Status.Key.Inserted;
   END_TRANSITION
   STEP "End production selected":   // S25, max time T#10S, warning time T#7S
   END_STEP
   TRANSITION Trans40 FROM "End production selected" TO END   // T40
      := NOT "AlwaysTRUE";
   END_TRANSITION
END_FUNCTION_BLOCK

FUNCTION "St1InsertionHandle" : Void
{ S7_Optimized_Access := 'TRUE' }
VERSION : 0.1
   VAR_TEMP 
      i : Int;
      res : Bool;
      empty : Bool;
      lastNOKIndex : Int;
   END_VAR


BEGIN
	
	#i := 1;
	"St1Insertion".SensorsState[#i] := "DevicesData".Camera[1].Result = 1;
	#i := #i + 1;
	"St1Insertion".SensorsState[#i] := "DevicesData".Camera[2].Result = 1;
	#i := #i + 1;
	"St1Insertion".SensorsState[#i] := "DevicesData".Camera[3].Result = 1;
	#i := #i + 1;
	"St1Insertion".SensorsState[#i] := "DevicesData".Camera[4].Result = 1;
	#i := #i + 1;
	"St1Insertion".SensorsState[#i] :=  "READER_MODEL_ACTUAL".ALL_SCANNER_OK = 1;
	#i := #i + 1;
	"St1Insertion".SensorsState[#i] :=  "SENSORES_LASER_OK" = 1;
	#i := #i + 1;
	"St1Insertion".SensorsState[#i] := FALSE;
	#i := #i + 1;
	"St1Insertion".SensorsState[#i] := FALSE;
	#i := #i + 1;
	"St1Insertion".SensorsState[#i] := FALSE;
	#i := #i + 1;
	"St1Insertion".SensorsState[#i] := FALSE;
	#i := #i + 1;
	"St1Insertion".SensorsState[#i] := FALSE;
	#i := #i + 1;
	"St1Insertion".SensorsState[#i] := FALSE;
	#i := #i + 1;
	"St1Insertion".SensorsState[#i] := FALSE;
	#i := #i + 1;
	"St1Insertion".SensorsState[#i] := FALSE;
	#i := #i + 1;
	"St1Insertion".SensorsState[#i] := FALSE;
	#i := #i + 1;
	"St1Insertion".SensorsState[#i] := FALSE;
	#i := #i + 1;
	"St1Insertion".SensorsState[#i] := FALSE;
	#i := #i + 1;
	"St1Insertion".SensorsState[#i] := FALSE;
	#i := #i + 1;
	"St1Insertion".SensorsState[#i] := FALSE;
	
	#lastNOKIndex := 1;
	
	#res := TRUE;
	#empty := true;
	FOR #i := 1 TO 20 DO
	    
	    //Check if all sensors are zero
	    IF "St1Insertion".SensorsState[#i] THEN
	        #empty := false;
	    END_IF;
	    //Check if sensor is correct
	    IF ("St1Insertion".SensorsState[#i] <> "St1Insertion".ExpectedSensors[#i]) AND
	            "St1Insertion".UsedSensors[#i] THEN
	            #res := false;
	            "St1Insertion".SensorsNOK[#i] := true;
	            "St1Insertion".NOKList[#lastNOKIndex] := #i;
	            #lastNOKIndex := #lastNOKIndex + 1;
	        ELSE
	            "St1Insertion".SensorsNOK[#i] := false;
	    END_IF;
	END_FOR;
	    
	//Reset rest of nok list
	FOR #i := #lastNOKIndex TO 20 DO
	        "St1Insertion".NOKList[#i] := 0;
	END_FOR;
	
	"St1Insertion".InsertionOK := #res;
	"St1Insertion".InsertionNOK := NOT #empty AND NOT #res;
	"St1Insertion".InsertionEmpty := #empty;
	
	
	
END_FUNCTION

FUNCTION_BLOCK "sq_carousel_st2"   // FB43, GRAPH
VERSION : 0.1
// stored: AcknowledgeErrorsRequired true, AutoNumber true, GraphVersion 6.0, InitialValuesAcquisition false, IsIECCheckEnabled false, LanguageInNetworks LAD, LockOperatingMode false, PermanentILProcessingInMANMode false, SetENOAutomatically false, SkipSteps false, UDAEnableTagReadback false, WithAlarmHandling true
   // inherited from GRAPH_BASE
   VAR
      OFF_SQ_BASE : Bool;
   END_VAR
   VAR_INPUT
      OFF_SQ { ExternalAccessible := 'False'; ExternalVisible := 'False'; ExternalWritable := 'False'} : Bool := false;   // Turn sequence off
      INIT_SQ { ExternalAccessible := 'False'; ExternalVisible := 'False'; ExternalWritable := 'False'} : Bool := false;   // Set sequence to initial state
      ACK_EF { ExternalAccessible := 'False'; ExternalVisible := 'False'; ExternalWritable := 'False'} : Bool := false;   // Acknowledge all errors and faults
      S_PREV { ExternalAccessible := 'False'; ExternalVisible := 'False'; ExternalWritable := 'False'} : Bool := false;   // Output previous step in parameter S_NO
      S_NEXT { ExternalAccessible := 'False'; ExternalVisible := 'False'; ExternalWritable := 'False'} : Bool := false;   // Indicate next step in parameter S_NO
      SW_AUTO { ExternalAccessible := 'False'; ExternalVisible := 'False'; ExternalWritable := 'False'} : Bool := false;   // Automatic mode
      SW_TAP { ExternalAccessible := 'False'; ExternalVisible := 'False'; ExternalWritable := 'False'} : Bool := false;   // Semiautomatic/switch with transition
      SW_TOP { ExternalAccessible := 'False'; ExternalVisible := 'False'; ExternalWritable := 'False'} : Bool := false;   // Semiautomatic/ignore transition
      SW_MAN { ExternalAccessible := 'False'; ExternalVisible := 'False'; ExternalWritable := 'False'} : Bool := false;   // Manual mode
      S_SEL { ExternalAccessible := 'False'; ExternalVisible := 'False'; ExternalWritable := 'False'} : Int := 0;   // Select step to be output to S_NO
      S_ON { ExternalAccessible := 'False'; ExternalVisible := 'False'; ExternalWritable := 'False'} : Bool := false;   // Activate step indicated in S_NO
      S_OFF { ExternalAccessible := 'False'; ExternalVisible := 'False'; ExternalWritable := 'False'} : Bool := false;   // Deactivate step indicated S_NO
      T_PUSH { ExternalAccessible := 'False'; ExternalVisible := 'False'; ExternalWritable := 'False'} : Bool := false;   // Enable transition to switch in semi automatic mode
   END_VAR
   VAR_OUTPUT
      S_NO { ExternalAccessible := 'False'; ExternalVisible := 'False'; ExternalWritable := 'False'} : Int := 0;   // Step number
      S_MORE { ExternalAccessible := 'False'; ExternalVisible := 'False'; ExternalWritable := 'False'} : Bool := false;   // More steps are available and can be shown in S_NO
      S_ACTIVE { ExternalAccessible := 'False'; ExternalVisible := 'False'; ExternalWritable := 'False'} : Bool := false;   // Step indicated in S_NO is active
      ERR_FLT { ExternalAccessible := 'False'; ExternalVisible := 'False'; ExternalWritable := 'False'} : Bool := false;   // Interlock or supervision group error
      AUTO_ON { ExternalAccessible := 'False'; ExternalVisible := 'False'; ExternalWritable := 'False'} : Bool := false;   // Automatic mode is active
      TAP_ON { ExternalAccessible := 'False'; ExternalVisible := 'False'; ExternalWritable := 'False'} : Bool := false;   // Semiautomatic mode/step with transition enabled
      TOP_ON { ExternalAccessible := 'False'; ExternalVisible := 'False'; ExternalWritable := 'False'} : Bool := false;   // Semiautomatic mode/ignore transition enabled
      MAN_ON { ExternalAccessible := 'False'; ExternalVisible := 'False'; ExternalWritable := 'False'} : Bool := false;   // Manual mode is active
   END_VAR
   VAR
      dummy : Bool;
      start : Bool;
      base : Bool;
   END_VAR
BEGIN
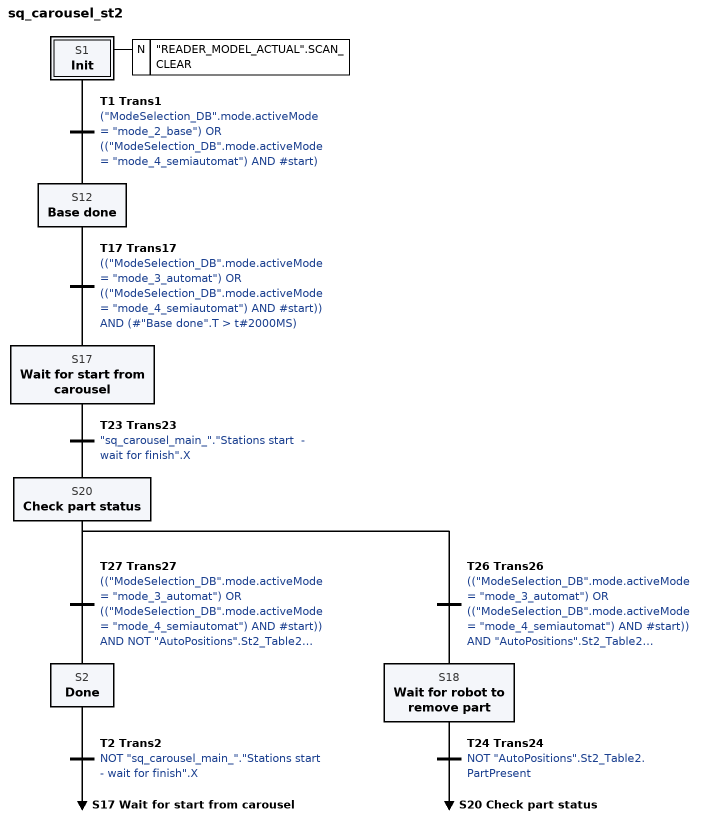
   // permanent pre-instructions
   NETWORK 1
   TITLE = base position
      #base := TRUE;

   // sequencer 1
   INITIAL_STEP Init:   // S1, max time T#10S, warning time T#7S
              N    "READER_MODEL_ACTUAL".SCAN_CLEAR
   END_STEP
   TRANSITION Trans1 FROM Init TO "Base done"   // T1
      := ("ModeSelection_DB".mode.activeMode = "mode_2_base") OR (("ModeSelection_DB".mode.activeMode = "mode_4_semiautomat") AND #start);
   END_TRANSITION
   STEP Done:   // S2, max time T#10S, warning time T#7S
   END_STEP
   TRANSITION Trans2 FROM Done TO "Wait for start from carousel"   // T2, jump
      := NOT "sq_carousel_main_"."Stations start  - wait for finish".X;
   END_TRANSITION
   STEP "Base done":   // S12, max time T#10S, warning time T#7S
   END_STEP
   TRANSITION Trans17 FROM "Base done" TO "Wait for start from carousel"   // T17
      := (("ModeSelection_DB".mode.activeMode = "mode_3_automat") OR (("ModeSelection_DB".mode.activeMode = "mode_4_semiautomat") AND #start)) AND (#"Base done".T > t#2000MS);
   END_TRANSITION
   STEP "Wait for start from carousel":   // S17, max time T#10S, warning time T#7S
   END_STEP
   TRANSITION Trans23 FROM "Wait for start from carousel" TO "Check part status"   // T23
      := "sq_carousel_main_"."Stations start  - wait for finish".X;
   END_TRANSITION
   STEP "Check part status":   // S20, max time T#10S, warning time T#7S
   END_STEP
   TRANSITION Trans27 FROM "Check part status" TO Done   // T27
      := (("ModeSelection_DB".mode.activeMode = "mode_3_automat") OR (("ModeSelection_DB".mode.activeMode = "mode_4_semiautomat") AND #start)) AND NOT "AutoPositions".St2_Table2.PartPresent AND "iR1OutOfSt2";
   END_TRANSITION
   TRANSITION Trans26 FROM "Check part status" TO "Wait for robot to remove part"   // T26
      := (("ModeSelection_DB".mode.activeMode = "mode_3_automat") OR (("ModeSelection_DB".mode.activeMode = "mode_4_semiautomat") AND #start)) AND "AutoPositions".St2_Table2.PartPresent;
   END_TRANSITION
   STEP "Wait for robot to remove part":   // S18, max time T#10S, warning time T#7S
   END_STEP
   TRANSITION Trans24 FROM "Wait for robot to remove part" TO "Check part status"   // T24, jump
      := NOT "AutoPositions".St2_Table2.PartPresent;
   END_TRANSITION
END_FUNCTION_BLOCK

FUNCTION_BLOCK "sq_jig"   // FB41, GRAPH
VERSION : 0.1
// stored: AcknowledgeErrorsRequired true, AutoNumber true, GraphVersion 6.0, InitialValuesAcquisition false, IsIECCheckEnabled false, LanguageInNetworks LAD, LockOperatingMode false, PermanentILProcessingInMANMode false, SetENOAutomatically false, SkipSteps false, UDAEnableTagReadback false, WithAlarmHandling true
   // inherited from GRAPH_BASE
   VAR
      OFF_SQ_BASE : Bool;
   END_VAR
   VAR_INPUT
      OFF_SQ { ExternalAccessible := 'False'; ExternalVisible := 'False'; ExternalWritable := 'False'} : Bool := false;   // Turn sequence off
      INIT_SQ { ExternalAccessible := 'False'; ExternalVisible := 'False'; ExternalWritable := 'False'} : Bool := false;   // Set sequence to initial state
      ACK_EF { ExternalAccessible := 'False'; ExternalVisible := 'False'; ExternalWritable := 'False'} : Bool := false;   // Acknowledge all errors and faults
      S_PREV { ExternalAccessible := 'False'; ExternalVisible := 'False'; ExternalWritable := 'False'} : Bool := false;   // Output previous step in parameter S_NO
      S_NEXT { ExternalAccessible := 'False'; ExternalVisible := 'False'; ExternalWritable := 'False'} : Bool := false;   // Indicate next step in parameter S_NO
      SW_AUTO { ExternalAccessible := 'False'; ExternalVisible := 'False'; ExternalWritable := 'False'} : Bool := false;   // Automatic mode
      SW_TAP { ExternalAccessible := 'False'; ExternalVisible := 'False'; ExternalWritable := 'False'} : Bool := false;   // Semiautomatic/switch with transition
      SW_TOP { ExternalAccessible := 'False'; ExternalVisible := 'False'; ExternalWritable := 'False'} : Bool := false;   // Semiautomatic/ignore transition
      SW_MAN { ExternalAccessible := 'False'; ExternalVisible := 'False'; ExternalWritable := 'False'} : Bool := false;   // Manual mode
      S_SEL { ExternalAccessible := 'False'; ExternalVisible := 'False'; ExternalWritable := 'False'} : Int := 0;   // Select step to be output to S_NO
      S_ON { ExternalAccessible := 'False'; ExternalVisible := 'False'; ExternalWritable := 'False'} : Bool := false;   // Activate step indicated in S_NO
      S_OFF { ExternalAccessible := 'False'; ExternalVisible := 'False'; ExternalWritable := 'False'} : Bool := false;   // Deactivate step indicated S_NO
      T_PUSH { ExternalAccessible := 'False'; ExternalVisible := 'False'; ExternalWritable := 'False'} : Bool := false;   // Enable transition to switch in semi automatic mode
   END_VAR
   VAR_OUTPUT
      S_NO { ExternalAccessible := 'False'; ExternalVisible := 'False'; ExternalWritable := 'False'} : Int := 0;   // Step number
      S_MORE { ExternalAccessible := 'False'; ExternalVisible := 'False'; ExternalWritable := 'False'} : Bool := false;   // More steps are available and can be shown in S_NO
      S_ACTIVE { ExternalAccessible := 'False'; ExternalVisible := 'False'; ExternalWritable := 'False'} : Bool := false;   // Step indicated in S_NO is active
      ERR_FLT { ExternalAccessible := 'False'; ExternalVisible := 'False'; ExternalWritable := 'False'} : Bool := false;   // Interlock or supervision group error
      AUTO_ON { ExternalAccessible := 'False'; ExternalVisible := 'False'; ExternalWritable := 'False'} : Bool := false;   // Automatic mode is active
      TAP_ON { ExternalAccessible := 'False'; ExternalVisible := 'False'; ExternalWritable := 'False'} : Bool := false;   // Semiautomatic mode/step with transition enabled
      TOP_ON { ExternalAccessible := 'False'; ExternalVisible := 'False'; ExternalWritable := 'False'} : Bool := false;   // Semiautomatic mode/ignore transition enabled
      MAN_ON { ExternalAccessible := 'False'; ExternalVisible := 'False'; ExternalWritable := 'False'} : Bool := false;   // Manual mode is active
   END_VAR
   VAR
      dummy : Bool;
      start : Bool;
      base : Bool;
   END_VAR
   VAR_TEMP   // added for the SCL form of the ladder/FBD networks
      _w1 : Bool;
   END_VAR
BEGIN
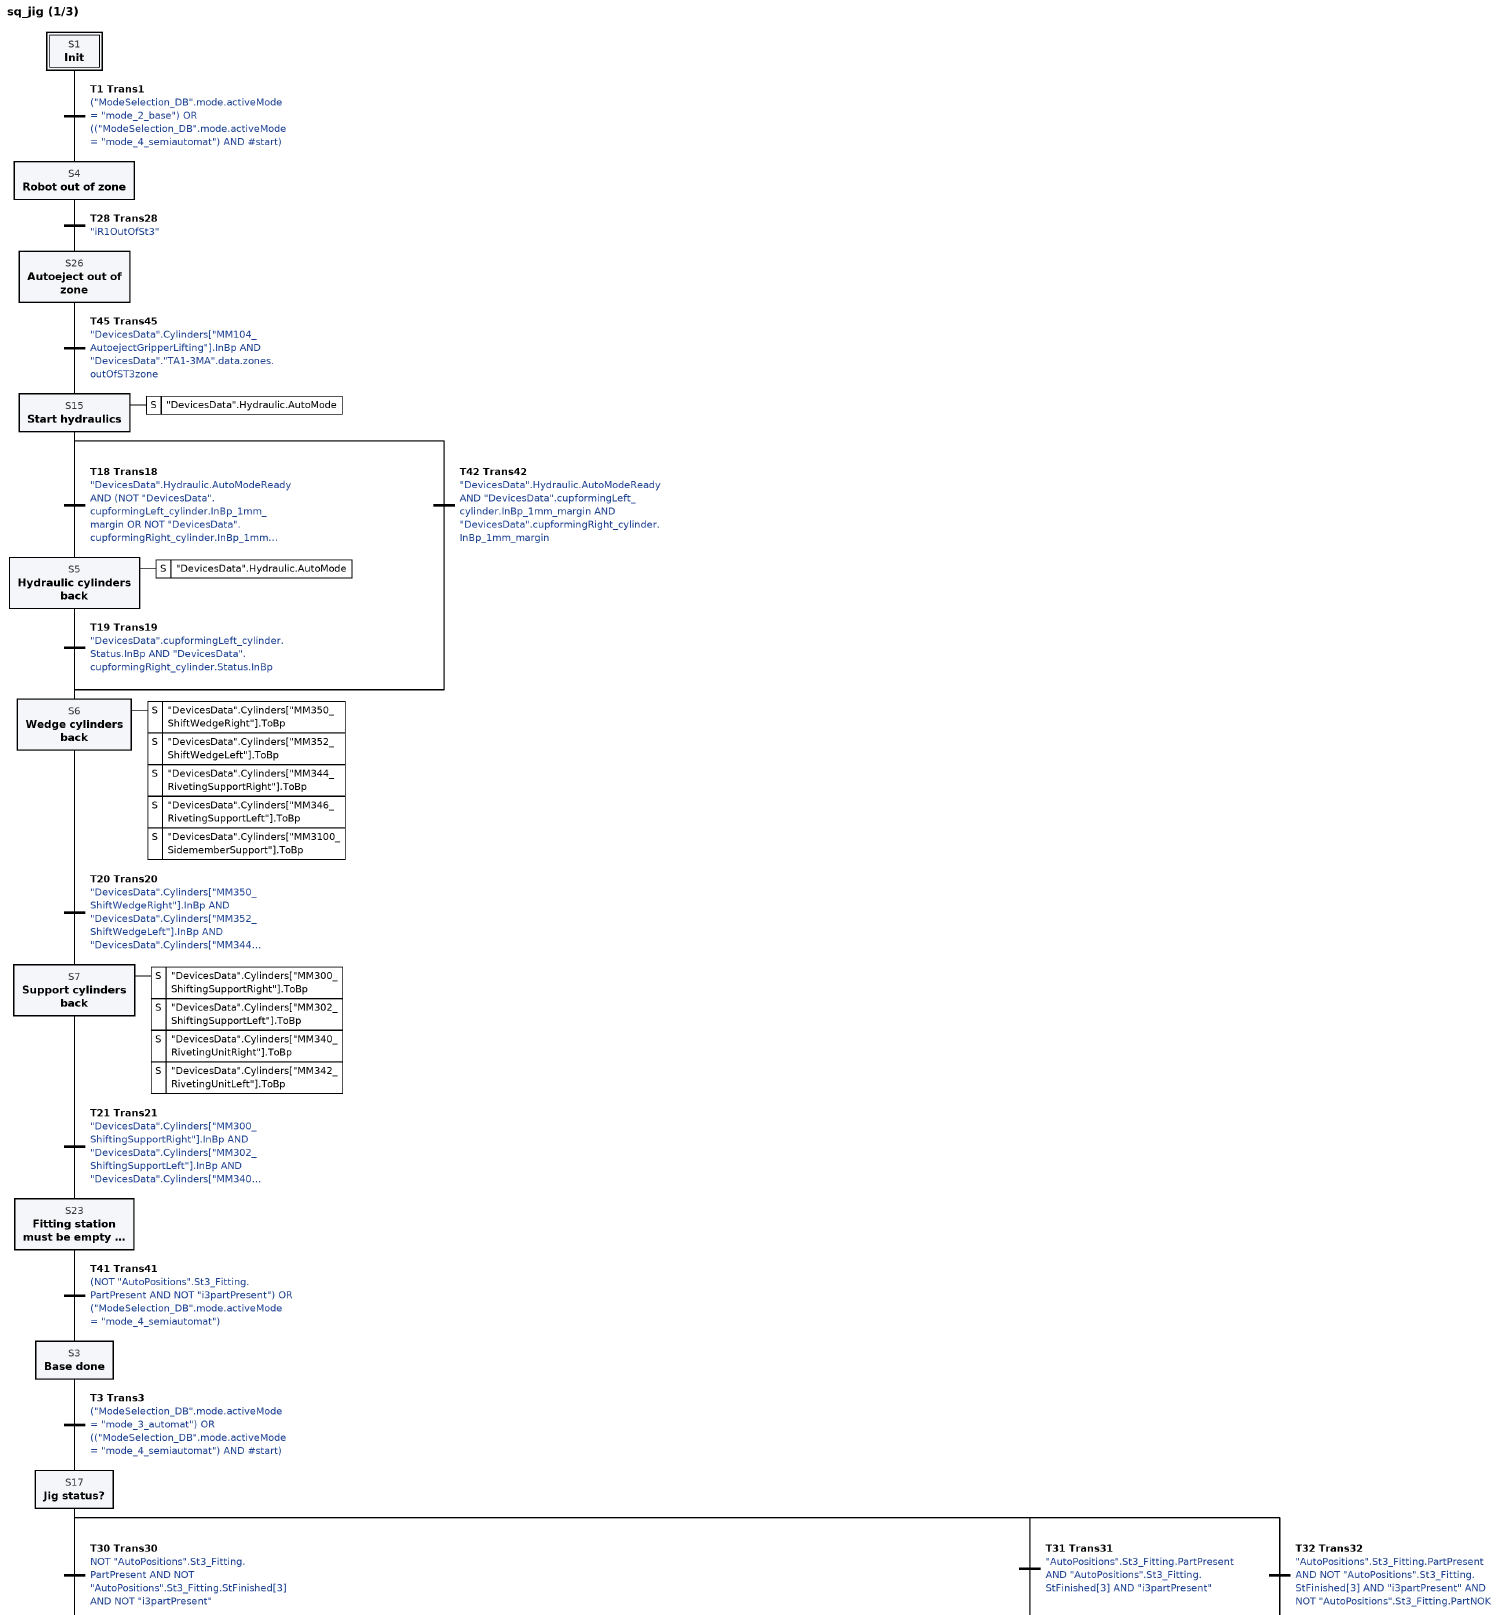
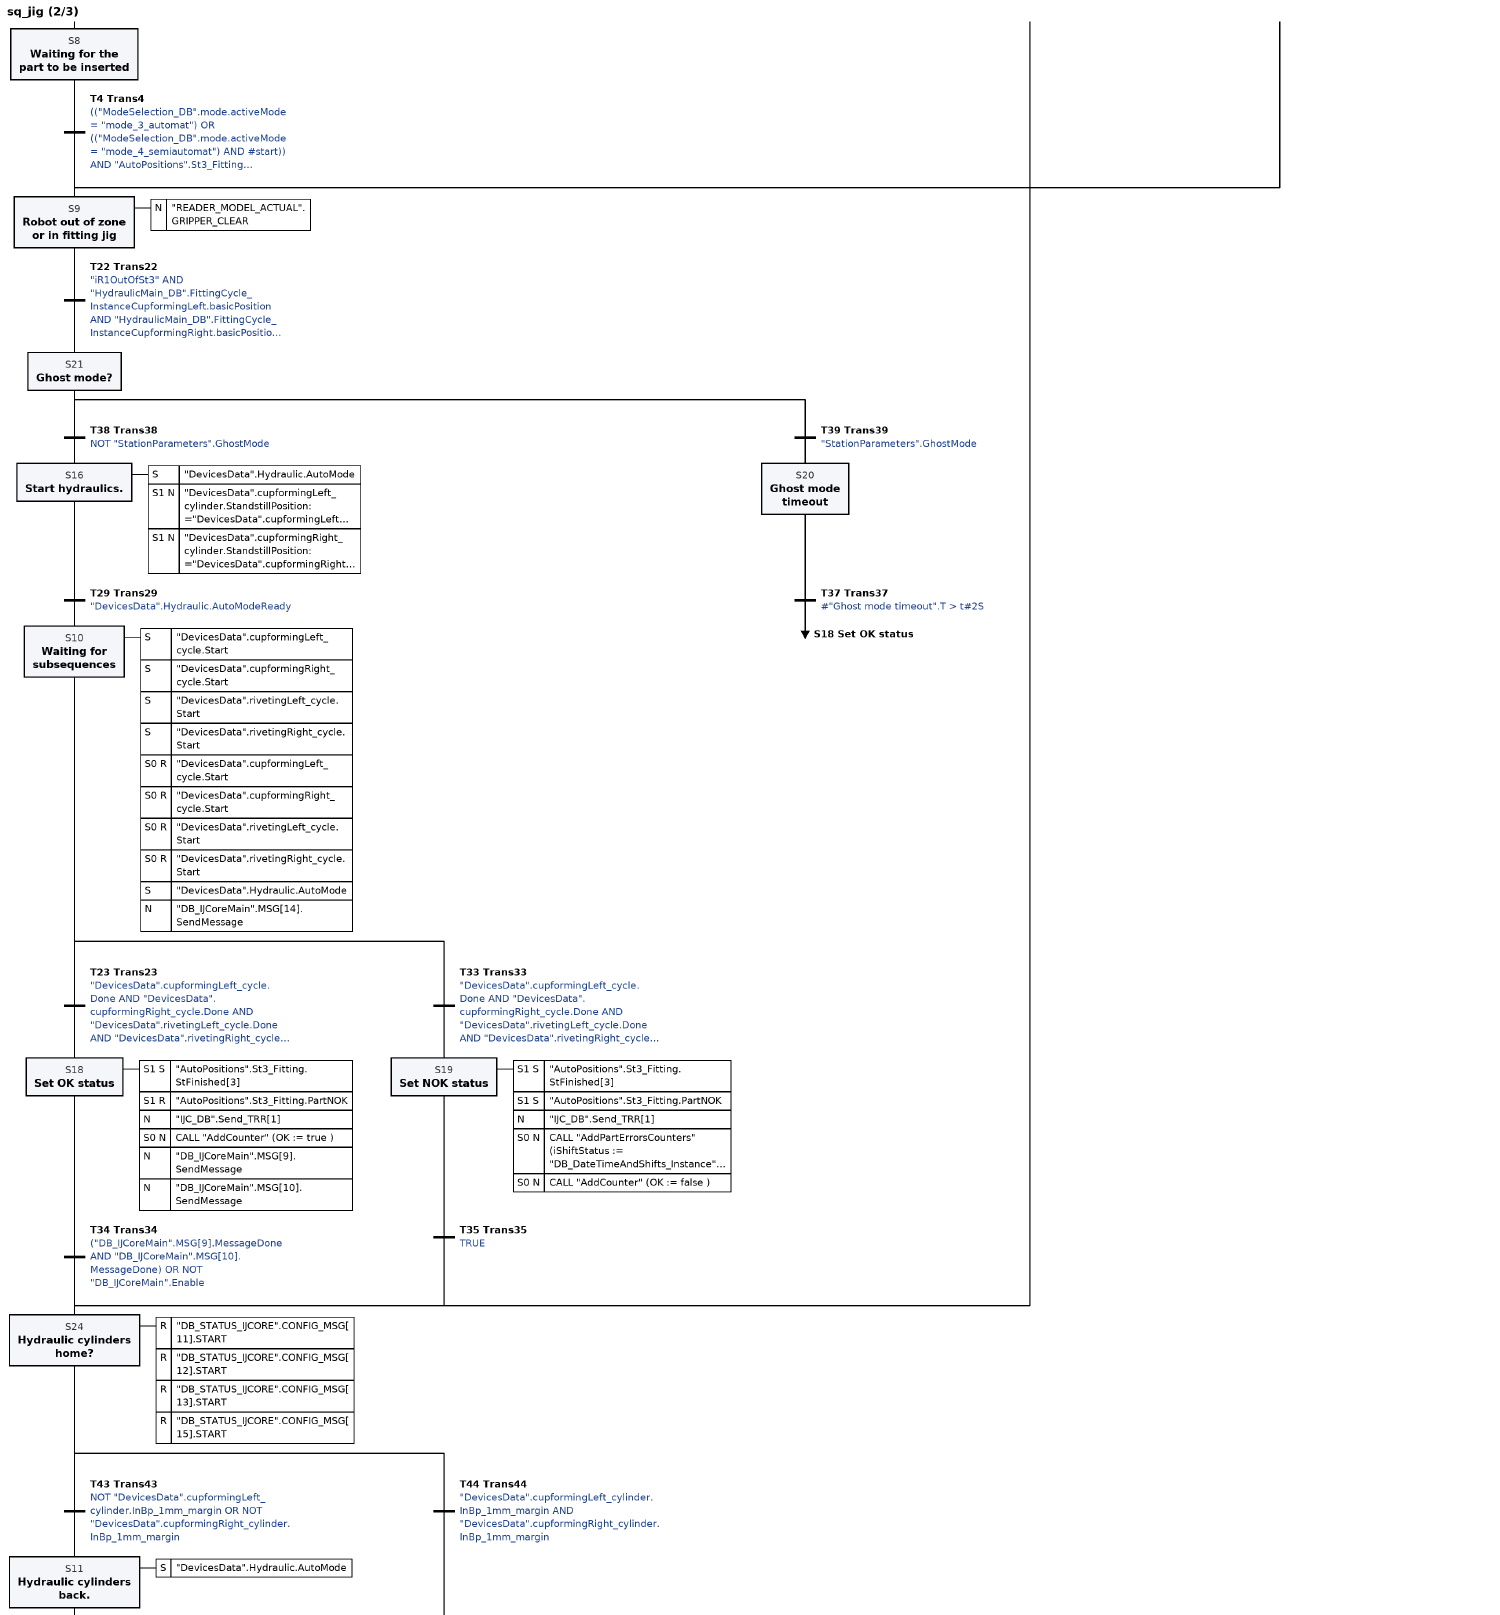
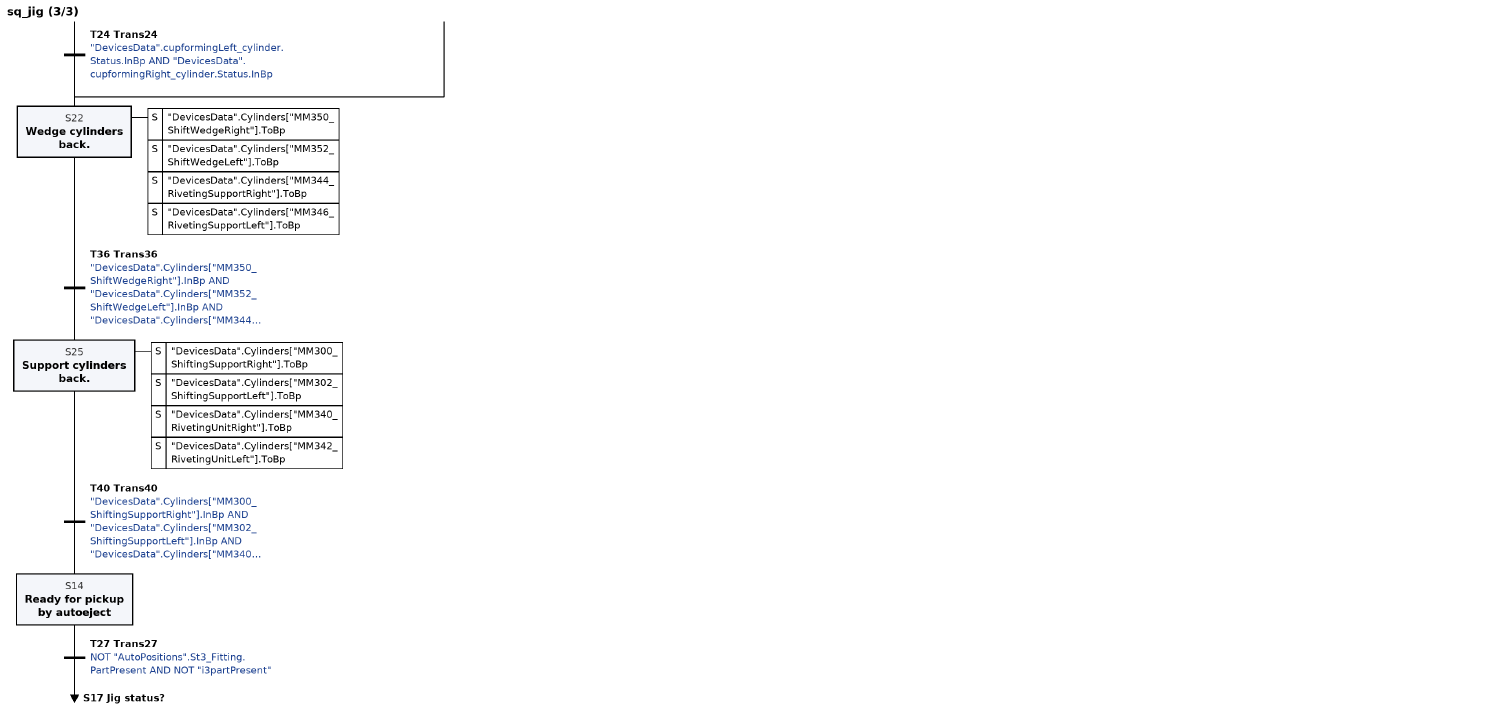
   // permanent pre-instructions
   NETWORK 1
   TITLE = base position
      #base := "HydraulicMain_DB".FittingCycle_InstanceCupformingLeft.basicPosition AND "HydraulicMain_DB".FittingCycle_InstanceCupformingRight.basicPosition AND "DB_Devices_Instance".RivetingCycleLeft_Instance.basicPosition AND "DB_Devices_Instance".RivetingCycleRight_Instance.basicPosition AND "DevicesData".Digiforce1.Ready AND "DevicesData".Digiforce1.programOK AND "DevicesData".Digiforce2.Ready AND "DevicesData".Digiforce2.programOK AND NOT "Devices_Diagnostic_DB".PNmissing;

   // sequencer 1
   INITIAL_STEP Init:   // S1, max time T#10S, warning time T#7S
   END_STEP
   TRANSITION Trans1 FROM Init TO "Robot out of zone"   // T1
      := ("ModeSelection_DB".mode.activeMode = "mode_2_base") OR (("ModeSelection_DB".mode.activeMode = "mode_4_semiautomat") AND #start);
   END_TRANSITION
   STEP "Start hydraulics":   // S15, max time T#10S, warning time T#7S
      supervision V := #"Start hydraulics".T > #"Start hydraulics".T_MAX;
              S    "DevicesData".Hydraulic.AutoMode
   END_STEP
   TRANSITION Trans18 FROM "Start hydraulics" TO "Hydraulic cylinders back"   // T18
      := "DevicesData".Hydraulic.AutoModeReady AND (NOT "DevicesData".cupformingLeft_cylinder.InBp_1mm_margin OR NOT "DevicesData".cupformingRight_cylinder.InBp_1mm_margin);
   END_TRANSITION
   TRANSITION Trans42 FROM "Start hydraulics" TO "Wedge cylinders back"   // T42
      := "DevicesData".Hydraulic.AutoModeReady AND "DevicesData".cupformingLeft_cylinder.InBp_1mm_margin AND "DevicesData".cupformingRight_cylinder.InBp_1mm_margin;
   END_TRANSITION
   STEP "Waiting for the part to be inserted":   // S8, max time T#10S, warning time T#7S
   END_STEP
   TRANSITION Trans4 FROM "Waiting for the part to be inserted" TO "Robot out of zone or in fitting jig"   // T4
      := (("ModeSelection_DB".mode.activeMode = "mode_3_automat") OR (("ModeSelection_DB".mode.activeMode = "mode_4_semiautomat") AND #start)) AND "AutoPositions".St3_Fitting.PartPresent AND NOT "AutoPositions".St3_Fitting.StFinished[3] AND ("i3partPresent" OR "StationParameters".GhostMode);
   END_TRANSITION
   STEP "Robot out of zone":   // S4, max time T#10S, warning time T#7S
      supervision V := #"Robot out of zone".T > #"Robot out of zone".T_MAX;
   END_STEP
   TRANSITION Trans28 FROM "Robot out of zone" TO "Autoeject out of zone"   // T28
      := "iR1OutOfSt3";
   END_TRANSITION
   STEP "Hydraulic cylinders back":   // S5, max time T#10S, warning time T#7S
      supervision V := #"Hydraulic cylinders back".T > #"Hydraulic cylinders back".T_MAX;
              S    "DevicesData".Hydraulic.AutoMode
   END_STEP
   TRANSITION Trans19 FROM "Hydraulic cylinders back" TO "Wedge cylinders back"   // T19
      := "DevicesData".cupformingLeft_cylinder.Status.InBp AND "DevicesData".cupformingRight_cylinder.Status.InBp;
   END_TRANSITION
   STEP "Wedge cylinders back":   // S6, max time T#10S, warning time T#7S
      supervision V := #"Wedge cylinders back".T > #"Wedge cylinders back".T_MAX;
              S    "DevicesData".Cylinders["MM350_ShiftWedgeRight"].ToBp
              S    "DevicesData".Cylinders["MM352_ShiftWedgeLeft"].ToBp
              S    "DevicesData".Cylinders["MM344_RivetingSupportRight"].ToBp
              S    "DevicesData".Cylinders["MM346_RivetingSupportLeft"].ToBp
              S    "DevicesData".Cylinders["MM3100_SidememberSupport"].ToBp
   END_STEP
   TRANSITION Trans20 FROM "Wedge cylinders back" TO "Support cylinders back"   // T20
      := "DevicesData".Cylinders["MM350_ShiftWedgeRight"].InBp AND "DevicesData".Cylinders["MM352_ShiftWedgeLeft"].InBp AND "DevicesData".Cylinders["MM344_RivetingSupportRight"].InBp AND "DevicesData".Cylinders["MM346_RivetingSupportLeft"].InBp AND "DevicesData".Cylinders["MM3100_SidememberSupport"].InBp;
   END_TRANSITION
   STEP "Support cylinders back":   // S7, max time T#10S, warning time T#7S
      supervision V := #"Support cylinders back".T > #"Support cylinders back".T_MAX;
              S    "DevicesData".Cylinders["MM300_ShiftingSupportRight"].ToBp
              S    "DevicesData".Cylinders["MM302_ShiftingSupportLeft"].ToBp
              S    "DevicesData".Cylinders["MM340_RivetingUnitRight"].ToBp
              S    "DevicesData".Cylinders["MM342_RivetingUnitLeft"].ToBp
   END_STEP
   TRANSITION Trans21 FROM "Support cylinders back" TO "Fitting station must be empty - remove part and delete status"   // T21
      := "DevicesData".Cylinders["MM300_ShiftingSupportRight"].InBp AND "DevicesData".Cylinders["MM302_ShiftingSupportLeft"].InBp AND "DevicesData".Cylinders["MM340_RivetingUnitRight"].InBp AND "DevicesData".Cylinders["MM342_RivetingUnitLeft"].InBp;
   END_TRANSITION
   STEP "Base done":   // S3, max time T#10S, warning time T#7S
   END_STEP
   TRANSITION Trans3 FROM "Base done" TO "Jig status?"   // T3
      := ("ModeSelection_DB".mode.activeMode = "mode_3_automat") OR (("ModeSelection_DB".mode.activeMode = "mode_4_semiautomat") AND #start);
   END_TRANSITION
   STEP "Robot out of zone or in fitting jig":   // S9, max time T#10S, warning time T#7S
      supervision V := #"Robot out of zone or in fitting jig".T > #"Robot out of zone or in fitting jig".T_MAX;
              N    "READER_MODEL_ACTUAL".GRIPPER_CLEAR
   END_STEP
   TRANSITION Trans22 FROM "Robot out of zone or in fitting jig" TO "Ghost mode?"   // T22
      := "iR1OutOfSt3" AND "HydraulicMain_DB".FittingCycle_InstanceCupformingLeft.basicPosition AND "HydraulicMain_DB".FittingCycle_InstanceCupformingRight.basicPosition AND "DB_Devices_Instance".RivetingCycleLeft_Instance.basicPosition AND "DB_Devices_Instance".RivetingCycleRight_Instance.basicPosition;
   END_TRANSITION
   STEP "Waiting for subsequences":   // S10, max time T#10S, warning time T#7S
              S    "DevicesData".cupformingLeft_cycle.Start
              S    "DevicesData".cupformingRight_cycle.Start
              S    "DevicesData".rivetingLeft_cycle.Start
              S    "DevicesData".rivetingRight_cycle.Start
          S0  R    "DevicesData".cupformingLeft_cycle.Start
          S0  R    "DevicesData".cupformingRight_cycle.Start
          S0  R    "DevicesData".rivetingLeft_cycle.Start
          S0  R    "DevicesData".rivetingRight_cycle.Start
              S    "DevicesData".Hydraulic.AutoMode
              N    "DB_IJCoreMain".MSG[14].SendMessage
   END_STEP
   TRANSITION Trans23 FROM "Waiting for subsequences" TO "Set OK status"   // T23
      := "DevicesData".cupformingLeft_cycle.Done AND "DevicesData".cupformingRight_cycle.Done AND "DevicesData".rivetingLeft_cycle.Done AND "DevicesData".rivetingRight_cycle.Done AND "DevicesData".cupformingLeft_cycle.OK AND "DevicesData".cupformingRight_cycle.OK AND "DevicesData".rivetingLeft_cycle.OK AND "DevicesData".rivetingRight_cycle.OK AND (("DB_IJCoreMain".MSG[14].MessageDone AND "DB_IJCoreMain".MSG[13].MessageDone AND ("DB_IJCoreMain".MSG[12].MessageDone OR "AlwaysTRUE")) OR NOT "DB_IJCoreMain".Enable) AND ("DB_IJCoreMain".MSG[15].MessageDone OR NOT "READER_MODEL_ACTUAL".PRODUCTO.NUM_TUBE);
   END_TRANSITION
   TRANSITION Trans33 FROM "Waiting for subsequences" TO "Set NOK status"   // T33
      := "DevicesData".cupformingLeft_cycle.Done AND "DevicesData".cupformingRight_cycle.Done AND "DevicesData".rivetingLeft_cycle.Done AND "DevicesData".rivetingRight_cycle.Done AND (("DB_IJCoreMain".MSG[14].MessageDone AND "DB_IJCoreMain".MSG[13].MessageDone AND ("DB_IJCoreMain".MSG[12].MessageDone OR "AlwaysTRUE")) OR NOT "DB_IJCoreMain".Enable) AND ("DB_IJCoreMain".MSG[15].MessageDone OR NOT "READER_MODEL_ACTUAL".PRODUCTO.NUM_TUBE);
   END_TRANSITION
   STEP "Hydraulic cylinders back.":   // S11, max time T#10S, warning time T#7S
      supervision V := #"Hydraulic cylinders back.".T > #"Hydraulic cylinders back.".T_MAX;
              S    "DevicesData".Hydraulic.AutoMode
   END_STEP
   TRANSITION Trans24 FROM "Hydraulic cylinders back." TO "Wedge cylinders back."   // T24
      := "DevicesData".cupformingLeft_cylinder.Status.InBp AND "DevicesData".cupformingRight_cylinder.Status.InBp;
   END_TRANSITION
   STEP "Autoeject out of zone":   // S26, max time T#10S, warning time T#7S
      supervision V := #"Autoeject out of zone".T > #"Autoeject out of zone".T_MAX;
   END_STEP
   TRANSITION Trans45 FROM "Autoeject out of zone" TO "Start hydraulics"   // T45
      := "DevicesData".Cylinders["MM104_AutoejectGripperLifting"].InBp AND "DevicesData"."TA1-3MA".data.zones.outOfST3zone;
   END_TRANSITION
   STEP "Ready for pickup by autoeject":   // S14, max time T#10S, warning time T#7S
   END_STEP
   TRANSITION Trans27 FROM "Ready for pickup by autoeject" TO "Jig status?"   // T27, jump
      := NOT "AutoPositions".St3_Fitting.PartPresent AND NOT "i3partPresent";
   END_TRANSITION
   STEP "Start hydraulics.":   // S16, max time T#10S, warning time T#7S
      supervision V := #"Start hydraulics.".T > #"Start hydraulics.".T_MAX;
              S    "DevicesData".Hydraulic.AutoMode
          S1  N    "DevicesData".cupformingLeft_cylinder.StandstillPosition:="DevicesData".cupformingLeft_cylinder.Position
          S1  N    "DevicesData".cupformingRight_cylinder.StandstillPosition:="DevicesData".cupformingRight_cylinder.Position
   END_STEP
   TRANSITION Trans29 FROM "Start hydraulics." TO "Waiting for subsequences"   // T29
      := "DevicesData".Hydraulic.AutoModeReady;
   END_TRANSITION
   STEP "Jig status?":   // S17, max time T#10S, warning time T#7S
   END_STEP
   TRANSITION Trans30 FROM "Jig status?" TO "Waiting for the part to be inserted"   // T30
      := NOT "AutoPositions".St3_Fitting.PartPresent AND NOT "AutoPositions".St3_Fitting.StFinished[3] AND NOT "i3partPresent";
   END_TRANSITION
   TRANSITION Trans31 FROM "Jig status?" TO "Hydraulic cylinders home?"   // T31
      := "AutoPositions".St3_Fitting.PartPresent AND "AutoPositions".St3_Fitting.StFinished[3] AND "i3partPresent";
   END_TRANSITION
   TRANSITION Trans32 FROM "Jig status?" TO "Robot out of zone or in fitting jig"   // T32
      := "AutoPositions".St3_Fitting.PartPresent AND NOT "AutoPositions".St3_Fitting.StFinished[3] AND "i3partPresent" AND NOT "AutoPositions".St3_Fitting.PartNOK;
   END_TRANSITION
   STEP "Set OK status":   // S18, max time T#10S, warning time T#7S
          S1  S    "AutoPositions".St3_Fitting.StFinished[3]
          S1  R    "AutoPositions".St3_Fitting.PartNOK
              N    "IJC_DB".Send_TRR[1]
          S0  N    CALL "AddCounter"
                   (OK := true
                   )
              N    "DB_IJCoreMain".MSG[9].SendMessage
              N    "DB_IJCoreMain".MSG[10].SendMessage
   END_STEP
   TRANSITION Trans34 FROM "Set OK status" TO "Hydraulic cylinders home?"   // T34
      := ("DB_IJCoreMain".MSG[9].MessageDone AND "DB_IJCoreMain".MSG[10].MessageDone) OR NOT "DB_IJCoreMain".Enable;
   END_TRANSITION
   STEP "Set NOK status":   // S19, max time T#10S, warning time T#7S
          S1  S    "AutoPositions".St3_Fitting.StFinished[3]
          S1  S    "AutoPositions".St3_Fitting.PartNOK
              N    "IJC_DB".Send_TRR[1]
          S0  N    CALL "AddPartErrorsCounters" (iShiftStatus := "DB_DateTimeAndShifts_Instance".ShiftStatus
                   )
          S0  N    CALL "AddCounter"
                   (OK := false
                   )
   END_STEP
   TRANSITION Trans35 FROM "Set NOK status" TO "Hydraulic cylinders home?"   // T35
      := TRUE;
   END_TRANSITION
   STEP "Ghost mode?":   // S21, max time T#10S, warning time T#7S
   END_STEP
   TRANSITION Trans38 FROM "Ghost mode?" TO "Start hydraulics."   // T38
      := NOT "StationParameters".GhostMode;
   END_TRANSITION
   TRANSITION Trans39 FROM "Ghost mode?" TO "Ghost mode timeout"   // T39
      := "StationParameters".GhostMode;
   END_TRANSITION
   STEP "Ghost mode timeout":   // S20, max time T#10S, warning time T#7S
   END_STEP
   TRANSITION Trans37 FROM "Ghost mode timeout" TO "Set OK status"   // T37, jump
      := #"Ghost mode timeout".T > t#2S;
   END_TRANSITION
   STEP "Fitting station must be empty - remove part and delete status":   // S23, max time T#2S, warning time T#7S
      supervision V := #"Fitting station must be empty - remove part and delete status".T > #"Fitting station must be empty - remove part and delete status".T_MAX;
   END_STEP
   TRANSITION Trans41 FROM "Fitting station must be empty - remove part and delete status" TO "Base done"   // T41
      := (NOT "AutoPositions".St3_Fitting.PartPresent AND NOT "i3partPresent") OR ("ModeSelection_DB".mode.activeMode = "mode_4_semiautomat");
   END_TRANSITION
   STEP "Hydraulic cylinders home?":   // S24, max time T#10S, warning time T#7S
              R    "DB_STATUS_IJCORE".CONFIG_MSG[11].START
              R    "DB_STATUS_IJCORE".CONFIG_MSG[12].START
              R    "DB_STATUS_IJCORE".CONFIG_MSG[13].START
              R    "DB_STATUS_IJCORE".CONFIG_MSG[15].START
   END_STEP
   TRANSITION Trans43 FROM "Hydraulic cylinders home?" TO "Hydraulic cylinders back."   // T43
      := NOT "DevicesData".cupformingLeft_cylinder.InBp_1mm_margin OR NOT "DevicesData".cupformingRight_cylinder.InBp_1mm_margin;
   END_TRANSITION
   TRANSITION Trans44 FROM "Hydraulic cylinders home?" TO "Wedge cylinders back."   // T44
      := "DevicesData".cupformingLeft_cylinder.InBp_1mm_margin AND "DevicesData".cupformingRight_cylinder.InBp_1mm_margin;
   END_TRANSITION
   STEP "Wedge cylinders back.":   // S22, max time T#10S, warning time T#7S
      supervision V := #"Wedge cylinders back.".T > #"Wedge cylinders back.".T_MAX;
              S    "DevicesData".Cylinders["MM350_ShiftWedgeRight"].ToBp
              S    "DevicesData".Cylinders["MM352_ShiftWedgeLeft"].ToBp
              S    "DevicesData".Cylinders["MM344_RivetingSupportRight"].ToBp
              S    "DevicesData".Cylinders["MM346_RivetingSupportLeft"].ToBp
   END_STEP
   TRANSITION Trans36 FROM "Wedge cylinders back." TO "Support cylinders back."   // T36
      := "DevicesData".Cylinders["MM350_ShiftWedgeRight"].InBp AND "DevicesData".Cylinders["MM352_ShiftWedgeLeft"].InBp AND "DevicesData".Cylinders["MM344_RivetingSupportRight"].InBp AND "DevicesData".Cylinders["MM346_RivetingSupportLeft"].InBp;
   END_TRANSITION
   STEP "Support cylinders back.":   // S25, max time T#10S, warning time T#7S
      supervision V := #"Support cylinders back.".T > #"Support cylinders back.".T_MAX;
              S    "DevicesData".Cylinders["MM300_ShiftingSupportRight"].ToBp
              S    "DevicesData".Cylinders["MM302_ShiftingSupportLeft"].ToBp
              S    "DevicesData".Cylinders["MM340_RivetingUnitRight"].ToBp
              S    "DevicesData".Cylinders["MM342_RivetingUnitLeft"].ToBp
   END_STEP
   TRANSITION Trans40 FROM "Support cylinders back." TO "Ready for pickup by autoeject"   // T40
      := "DevicesData".Cylinders["MM300_ShiftingSupportRight"].InBp AND "DevicesData".Cylinders["MM302_ShiftingSupportLeft"].InBp AND "DevicesData".Cylinders["MM340_RivetingUnitRight"].InBp AND "DevicesData".Cylinders["MM342_RivetingUnitLeft"].InBp;
   END_TRANSITION

   // permanent post-instructions
   NETWORK 1
   TITLE = Hydraulic cylinders back
      #_w1 := #"Hydraulic cylinders back".X OR #"Hydraulic cylinders back.".X;
      IF #_w1 AND NOT "DevicesData".cupformingLeft_cylinder.Status.InBp THEN
          "DevicesData".cupformingLeft_cylinder.Status.ToBp := TRUE;
      END_IF;
      IF #_w1 AND NOT "DevicesData".cupformingRight_cylinder.Status.InBp THEN
          "DevicesData".cupformingRight_cylinder.Status.ToBp := TRUE;
      END_IF;
      IF #_w1 AND "DevicesData".cupformingLeft_cylinder.Status.InBp THEN
          "DevicesData".cupformingLeft_cylinder.Status.ToBp := FALSE;
      END_IF;
      IF #_w1 AND "DevicesData".cupformingRight_cylinder.Status.InBp THEN
          "DevicesData".cupformingRight_cylinder.Status.ToBp := FALSE;
      END_IF;
END_FUNCTION_BLOCK

FUNCTION_BLOCK "sq_manipulator"   // FB44, GRAPH
VERSION : 0.1
// stored: AcknowledgeErrorsRequired true, AutoNumber true, GraphVersion 6.0, InitialValuesAcquisition false, IsIECCheckEnabled false, LanguageInNetworks LAD, LockOperatingMode false, PermanentILProcessingInMANMode false, SetENOAutomatically false, SkipSteps false, UDAEnableTagReadback false, WithAlarmHandling true
   // inherited from GRAPH_BASE
   VAR
      OFF_SQ_BASE : Bool;
   END_VAR
   VAR_INPUT
      OFF_SQ { ExternalAccessible := 'False'; ExternalVisible := 'False'; ExternalWritable := 'False'} : Bool := false;   // Turn sequence off
      INIT_SQ { ExternalAccessible := 'False'; ExternalVisible := 'False'; ExternalWritable := 'False'} : Bool := false;   // Set sequence to initial state
      ACK_EF { ExternalAccessible := 'False'; ExternalVisible := 'False'; ExternalWritable := 'False'} : Bool := false;   // Acknowledge all errors and faults
      S_PREV { ExternalAccessible := 'False'; ExternalVisible := 'False'; ExternalWritable := 'False'} : Bool := false;   // Output previous step in parameter S_NO
      S_NEXT { ExternalAccessible := 'False'; ExternalVisible := 'False'; ExternalWritable := 'False'} : Bool := false;   // Indicate next step in parameter S_NO
      SW_AUTO { ExternalAccessible := 'False'; ExternalVisible := 'False'; ExternalWritable := 'False'} : Bool := false;   // Automatic mode
      SW_TAP { ExternalAccessible := 'False'; ExternalVisible := 'False'; ExternalWritable := 'False'} : Bool := false;   // Semiautomatic/switch with transition
      SW_TOP { ExternalAccessible := 'False'; ExternalVisible := 'False'; ExternalWritable := 'False'} : Bool := false;   // Semiautomatic/ignore transition
      SW_MAN { ExternalAccessible := 'False'; ExternalVisible := 'False'; ExternalWritable := 'False'} : Bool := false;   // Manual mode
      S_SEL { ExternalAccessible := 'False'; ExternalVisible := 'False'; ExternalWritable := 'False'} : Int := 0;   // Select step to be output to S_NO
      S_ON { ExternalAccessible := 'False'; ExternalVisible := 'False'; ExternalWritable := 'False'} : Bool := false;   // Activate step indicated in S_NO
      S_OFF { ExternalAccessible := 'False'; ExternalVisible := 'False'; ExternalWritable := 'False'} : Bool := false;   // Deactivate step indicated S_NO
      T_PUSH { ExternalAccessible := 'False'; ExternalVisible := 'False'; ExternalWritable := 'False'} : Bool := false;   // Enable transition to switch in semi automatic mode
   END_VAR
   VAR_OUTPUT
      S_NO { ExternalAccessible := 'False'; ExternalVisible := 'False'; ExternalWritable := 'False'} : Int := 0;   // Step number
      S_MORE { ExternalAccessible := 'False'; ExternalVisible := 'False'; ExternalWritable := 'False'} : Bool := false;   // More steps are available and can be shown in S_NO
      S_ACTIVE { ExternalAccessible := 'False'; ExternalVisible := 'False'; ExternalWritable := 'False'} : Bool := false;   // Step indicated in S_NO is active
      ERR_FLT { ExternalAccessible := 'False'; ExternalVisible := 'False'; ExternalWritable := 'False'} : Bool := false;   // Interlock or supervision group error
      AUTO_ON { ExternalAccessible := 'False'; ExternalVisible := 'False'; ExternalWritable := 'False'} : Bool := false;   // Automatic mode is active
      TAP_ON { ExternalAccessible := 'False'; ExternalVisible := 'False'; ExternalWritable := 'False'} : Bool := false;   // Semiautomatic mode/step with transition enabled
      TOP_ON { ExternalAccessible := 'False'; ExternalVisible := 'False'; ExternalWritable := 'False'} : Bool := false;   // Semiautomatic mode/ignore transition enabled
      MAN_ON { ExternalAccessible := 'False'; ExternalVisible := 'False'; ExternalWritable := 'False'} : Bool := false;   // Manual mode is active
   END_VAR
   VAR
      dummy : Bool;
      start : Bool;
      base : Bool;
      IEC_Timer_0_Instance { S7_SetPoint := 'True'} : TON_TIME;
      IEC_Timer_0_Instance_1 { S7_SetPoint := 'True'} : TON_TIME;
      IEC_Timer_0_Instance_2 { S7_SetPoint := 'True'} : TON_TIME;
   END_VAR
BEGIN
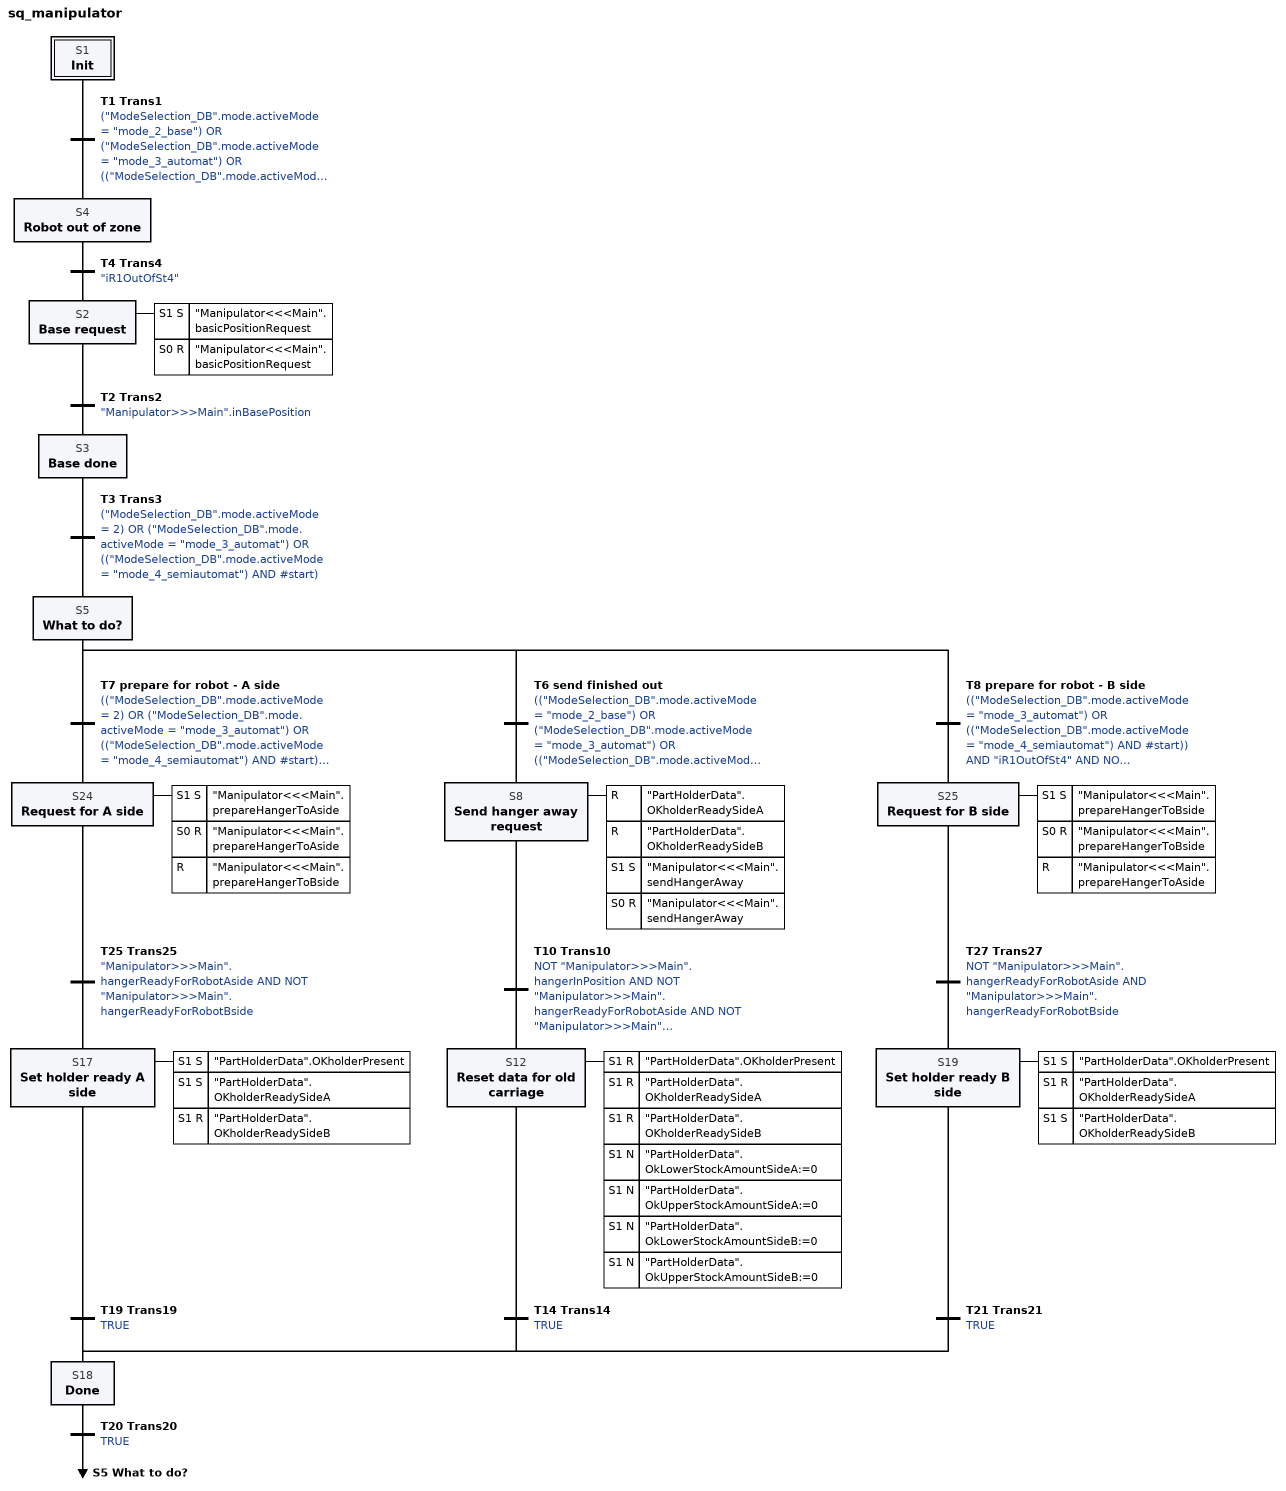
   // permanent pre-instructions
   NETWORK 1
   TITLE = base
      #base := #"Base done".X;

   // sequencer 1
   INITIAL_STEP Init:   // S1, max time T#10S, warning time T#7S
   END_STEP
   TRANSITION Trans1 FROM Init TO "Robot out of zone"   // T1
      := ("ModeSelection_DB".mode.activeMode = "mode_2_base") OR ("ModeSelection_DB".mode.activeMode = "mode_3_automat") OR (("ModeSelection_DB".mode.activeMode = "mode_4_semiautomat") AND #start);
   END_TRANSITION
   STEP "Base request":   // S2, max time T#10S, warning time T#7S
          S1  S    "Manipulator<<<Main".basicPositionRequest
          S0  R    "Manipulator<<<Main".basicPositionRequest
   END_STEP
   TRANSITION Trans2 FROM "Base request" TO "Base done"   // T2
      := "Manipulator>>>Main".inBasePosition;
   END_TRANSITION
   STEP "Base done":   // S3, max time T#10S, warning time T#7S
   END_STEP
   TRANSITION Trans3 FROM "Base done" TO "What to do?"   // T3
      := ("ModeSelection_DB".mode.activeMode = 2) OR ("ModeSelection_DB".mode.activeMode = "mode_3_automat") OR (("ModeSelection_DB".mode.activeMode = "mode_4_semiautomat") AND #start);
   END_TRANSITION
   STEP "Robot out of zone":   // S4, max time T#10S, warning time T#7S
      supervision V := (#"Robot out of zone".T > #"Robot out of zone".T_MAX) AND (T#0MS > #"Robot out of zone".T_MAX);
   END_STEP
   TRANSITION Trans4 FROM "Robot out of zone" TO "Base request"   // T4
      := "iR1OutOfSt4";
   END_TRANSITION
   STEP "What to do?":   // S5, max time T#10S, warning time T#7S
   END_STEP
   TRANSITION "prepare for robot - A side" FROM "What to do?" TO "Request for A side"   // T7
      := (("ModeSelection_DB".mode.activeMode = 2) OR ("ModeSelection_DB".mode.activeMode = "mode_3_automat") OR (("ModeSelection_DB".mode.activeMode = "mode_4_semiautomat") AND #start)) AND "iR1OutOfSt4" AND NOT "PartHolderData".OKholderReadySideA AND (("PartHolderData".OkLowerStockAmountSideA < "StationParameters".OKLowerStockSize) OR ("PartHolderData".OkUpperStockAmountSideA < "StationParameters".OKUpperStockSize));
   END_TRANSITION
   TRANSITION "send finished out" FROM "What to do?" TO "Send hanger away request"   // T6
      := (("ModeSelection_DB".mode.activeMode = "mode_2_base") OR ("ModeSelection_DB".mode.activeMode = "mode_3_automat") OR (("ModeSelection_DB".mode.activeMode = "mode_4_semiautomat") AND #start)) AND "iR1OutOfSt4" AND "PartHolderData".OKholderPresent AND ((("PartHolderData".OkLowerStockAmountSideA >= "StationParameters".OKLowerStockSize) AND ("PartHolderData".OkUpperStockAmountSideA >= "StationParameters".OKUpperStockSize) AND ("PartHolderData".OkLowerStockAmountSideB >= "StationParameters".OKLowerStockSize) AND ("PartHolderData".OkUpperStockAmountSideB >= "StationParameters".OKUpperStockSize)) OR "Manipulator<<<Main".reserve[0].%X0) AND NOT "sq_robot_"."Dropoff part to manipulator level1".X AND NOT "sq_robot_"."Dropoff part to manipulator level2".X;
   END_TRANSITION
   TRANSITION "prepare for robot - B side" FROM "What to do?" TO "Request for B side"   // T8
      := (("ModeSelection_DB".mode.activeMode = "mode_3_automat") OR (("ModeSelection_DB".mode.activeMode = "mode_4_semiautomat") AND #start)) AND "iR1OutOfSt4" AND NOT "PartHolderData".OKholderReadySideB AND (("PartHolderData".OkLowerStockAmountSideB < "StationParameters".OKLowerStockSize) OR ("PartHolderData".OkUpperStockAmountSideB < "StationParameters".OKUpperStockSize)) AND ("PartHolderData".OkLowerStockAmountSideA >= "StationParameters".OKLowerStockSize) AND ("PartHolderData".OkUpperStockAmountSideA >= "StationParameters".OKUpperStockSize);
   END_TRANSITION
   STEP "Request for B side":   // S25, max time T#30S, warning time T#7S
      supervision V := (#"Request for B side".T > #"Request for B side".T_MAX) AND (T#0MS > #"Request for B side".T_MAX);
          S1  S    "Manipulator<<<Main".prepareHangerToBside
          S0  R    "Manipulator<<<Main".prepareHangerToBside
              R    "Manipulator<<<Main".prepareHangerToAside
   END_STEP
   TRANSITION Trans27 FROM "Request for B side" TO "Set holder ready B side"   // T27
      := NOT "Manipulator>>>Main".hangerReadyForRobotAside AND "Manipulator>>>Main".hangerReadyForRobotBside;
   END_TRANSITION
   STEP "Set holder ready A side":   // S17, max time T#10S, warning time T#7S
          S1  S    "PartHolderData".OKholderPresent
          S1  S    "PartHolderData".OKholderReadySideA
          S1  R    "PartHolderData".OKholderReadySideB
   END_STEP
   TRANSITION Trans19 FROM "Set holder ready A side" TO Done   // T19
      := TRUE;
   END_TRANSITION
   STEP Done:   // S18, max time T#10S, warning time T#7S
   END_STEP
   TRANSITION Trans20 FROM Done TO "What to do?"   // T20, jump
      := TRUE;
   END_TRANSITION
   STEP "Send hanger away request":   // S8, max time T#10S, warning time T#7S
              R    "PartHolderData".OKholderReadySideA
              R    "PartHolderData".OKholderReadySideB
          S1  S    "Manipulator<<<Main".sendHangerAway
          S0  R    "Manipulator<<<Main".sendHangerAway
   END_STEP
   TRANSITION Trans10 FROM "Send hanger away request" TO "Reset data for old carriage"   // T10
      := NOT "Manipulator>>>Main".hangerInPosition AND NOT "Manipulator>>>Main".hangerReadyForRobotAside AND NOT "Manipulator>>>Main".hangerReadyForRobotBside;
   END_TRANSITION
   STEP "Set holder ready B side":   // S19, max time T#10S, warning time T#7S
          S1  S    "PartHolderData".OKholderPresent
          S1  R    "PartHolderData".OKholderReadySideA
          S1  S    "PartHolderData".OKholderReadySideB
   END_STEP
   TRANSITION Trans21 FROM "Set holder ready B side" TO Done   // T21
      := TRUE;
   END_TRANSITION
   STEP "Reset data for old carriage":   // S12, max time T#10S, warning time T#7S
          S1  R    "PartHolderData".OKholderPresent
          S1  R    "PartHolderData".OKholderReadySideA
          S1  R    "PartHolderData".OKholderReadySideB
          S1  N    "PartHolderData".OkLowerStockAmountSideA:=0
          S1  N    "PartHolderData".OkUpperStockAmountSideA:=0
          S1  N    "PartHolderData".OkLowerStockAmountSideB:=0
          S1  N    "PartHolderData".OkUpperStockAmountSideB:=0
   END_STEP
   TRANSITION Trans14 FROM "Reset data for old carriage" TO Done   // T14
      := TRUE;
   END_TRANSITION
   STEP "Request for A side":   // S24, max time T#30S, warning time T#7S
      supervision V := (#"Request for A side".T > #"Request for A side".T_MAX) AND (T#0MS > #"Request for A side".T_MAX);
          S1  S    "Manipulator<<<Main".prepareHangerToAside
          S0  R    "Manipulator<<<Main".prepareHangerToAside
              R    "Manipulator<<<Main".prepareHangerToBside
   END_STEP
   TRANSITION Trans25 FROM "Request for A side" TO "Set holder ready A side"   // T25
      := "Manipulator>>>Main".hangerReadyForRobotAside AND NOT "Manipulator>>>Main".hangerReadyForRobotBside;
   END_TRANSITION
END_FUNCTION_BLOCK

FUNCTION_BLOCK "sq_robot"   // FB42, GRAPH
VERSION : 0.1
// stored: AcknowledgeErrorsRequired true, AutoNumber true, GraphVersion 6.0, InitialValuesAcquisition false, IsIECCheckEnabled false, LanguageInNetworks LAD, LockOperatingMode false, PermanentILProcessingInMANMode false, SetENOAutomatically false, SkipSteps false, UDAEnableTagReadback false, WithAlarmHandling true
   // inherited from GRAPH_BASE
   VAR
      OFF_SQ_BASE : Bool;
   END_VAR
   VAR_INPUT
      OFF_SQ { ExternalWritable := 'False'} : Bool := false;   // Turn sequence off
      INIT_SQ { ExternalWritable := 'False'} : Bool := false;   // Set sequence to initial state
      ACK_EF { ExternalWritable := 'False'} : Bool := false;   // Acknowledge all errors and faults
      S_PREV { ExternalWritable := 'False'} : Bool := false;   // Output previous step in parameter S_NO
      S_NEXT { ExternalWritable := 'False'} : Bool := false;   // Indicate next step in parameter S_NO
      SW_AUTO { ExternalWritable := 'False'} : Bool := false;   // Automatic mode
      SW_TAP { ExternalWritable := 'False'} : Bool := false;   // Semiautomatic/switch with transition
      SW_TOP { ExternalWritable := 'False'} : Bool := false;   // Semiautomatic/ignore transition
      SW_MAN { ExternalWritable := 'False'} : Bool := false;   // Manual mode
      S_SEL { ExternalWritable := 'False'} : Int := 0;   // Select step to be output to S_NO
      S_ON { ExternalWritable := 'False'} : Bool := false;   // Activate step indicated in S_NO
      S_OFF { ExternalWritable := 'False'} : Bool := false;   // Deactivate step indicated S_NO
      T_PUSH { ExternalWritable := 'False'} : Bool := false;   // Enable transition to switch in semi automatic mode
   END_VAR
   VAR_OUTPUT
      S_NO { ExternalWritable := 'False'} : Int := 0;   // Step number
      S_MORE { ExternalWritable := 'False'} : Bool := false;   // More steps are available and can be shown in S_NO
      S_ACTIVE { ExternalWritable := 'False'} : Bool := false;   // Step indicated in S_NO is active
      ERR_FLT { ExternalWritable := 'False'} : Bool := false;   // Interlock or supervision group error
      AUTO_ON { ExternalWritable := 'False'} : Bool := false;   // Automatic mode is active
      TAP_ON { ExternalWritable := 'False'} : Bool := false;   // Semiautomatic mode/step with transition enabled
      TOP_ON { ExternalWritable := 'False'} : Bool := false;   // Semiautomatic mode/ignore transition enabled
      MAN_ON { ExternalWritable := 'False'} : Bool := false;   // Manual mode is active
   END_VAR
   VAR
      dummy : Bool;
      start : Bool;
      base : Bool;
      startMastering : Bool;
      startBraketest : Bool;
      prgNrForManipulatorDropoff : Byte;
   END_VAR
   VAR CONSTANT
      jobHoming : Byte := 1;
      jobCarouselPickup : Byte := 2;
      jobJigDropoff : Byte := 3;
      jobAutoEjectPickup : Byte := 4;
      jobMastering : Byte := 10;
      jobBreaktest : Byte := 11;
      jobManipulatorDropoff1 : Byte := 21;   // top far
      jobManipulatorDropoff2 : Byte := 22;   // top middle
      jobManipulatorDropoff3 : Byte := 23;   // top near
      jobManipulatorDropoff4 : Byte := 24;   // bottom far
      jobManipulatorDropoff5 : Byte := 25;   // bottom middle
      jobManipulatorDropoff6 : Byte := 26;   // bottom near
      jobManipulatorForTesting : Byte := 30;
   END_VAR
   VAR_TEMP   // added for the SCL form of the ladder/FBD networks
      _w1 : Bool;
      _w2 : Bool;
   END_VAR
BEGIN
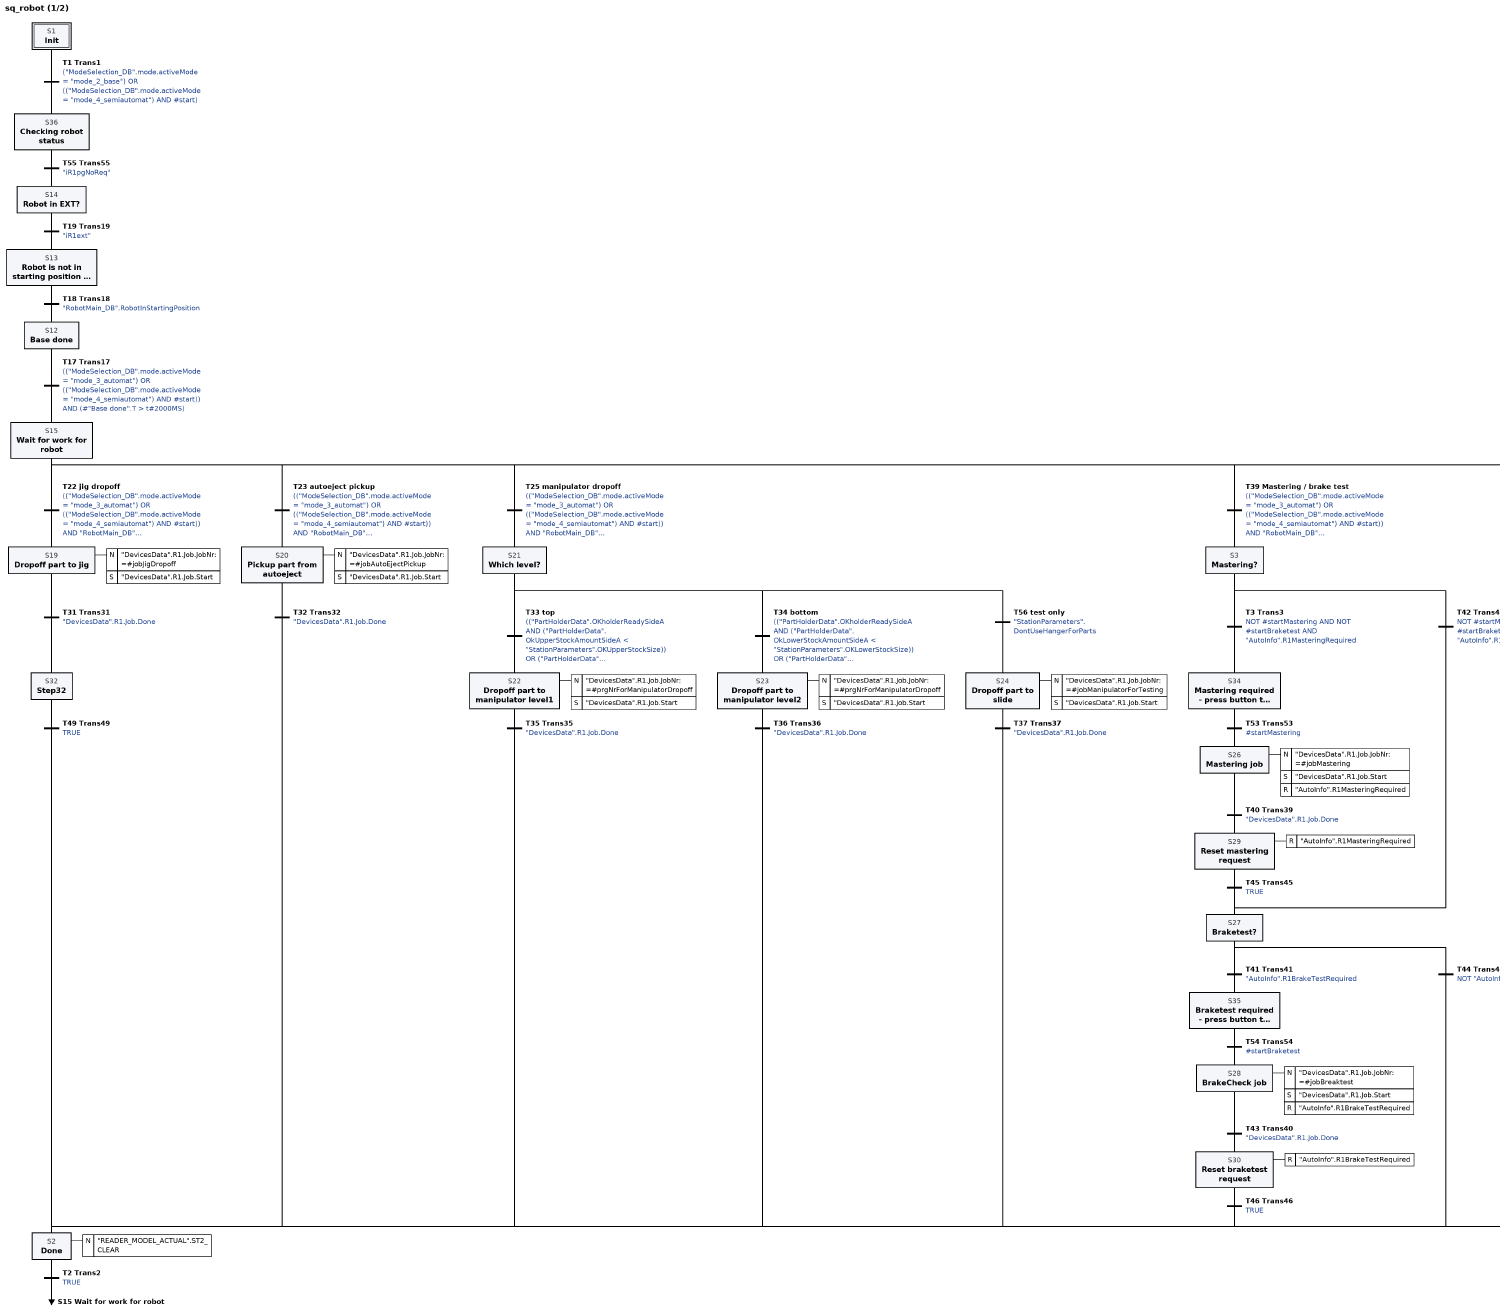
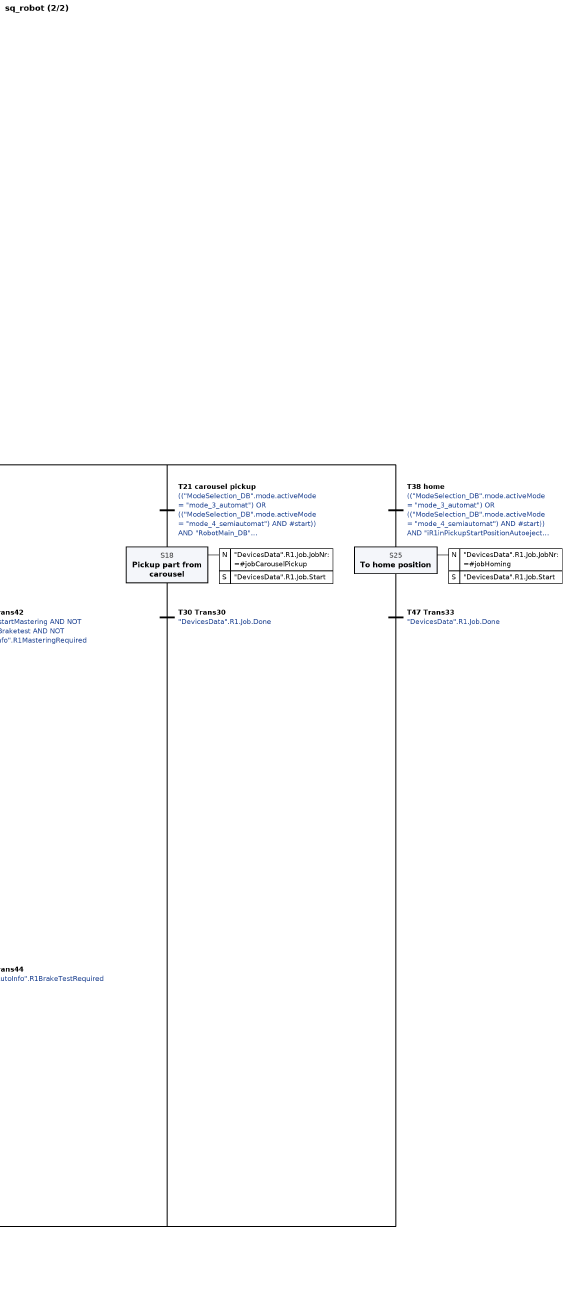
   // permanent pre-instructions
   NETWORK 1
   TITLE = prg for top level
      #_w1 := #"Dropoff part to manipulator level1".S1 AND "PartHolderData".OKholderReadySideA AND NOT "PartHolderData".OKholderReadySideB;
      IF #_w1 AND ("PartHolderData".OkUpperStockAmountSideA = 0) THEN
          #prgNrForManipulatorDropoff := #jobManipulatorDropoff1;
      END_IF;
      IF #_w1 AND ("PartHolderData".OkUpperStockAmountSideA = 1) THEN
          #prgNrForManipulatorDropoff := #jobManipulatorDropoff2;
      END_IF;
      IF #_w1 AND ("PartHolderData".OkUpperStockAmountSideA = 2) THEN
          #prgNrForManipulatorDropoff := #jobManipulatorDropoff3;
      END_IF;
      #_w2 := #"Dropoff part to manipulator level1".S1 AND NOT "PartHolderData".OKholderReadySideA AND "PartHolderData".OKholderReadySideB;
      IF #_w2 AND ("PartHolderData".OkUpperStockAmountSideB = 0) THEN
          #prgNrForManipulatorDropoff := #jobManipulatorDropoff1;
      END_IF;
      IF #_w2 AND ("PartHolderData".OkUpperStockAmountSideB = 1) THEN
          #prgNrForManipulatorDropoff := #jobManipulatorDropoff2;
      END_IF;
      IF #_w2 AND ("PartHolderData".OkUpperStockAmountSideB = 2) THEN
          #prgNrForManipulatorDropoff := #jobManipulatorDropoff3;
      END_IF;
   NETWORK 2
   TITLE = prg for bottom level
      #_w1 := #"Dropoff part to manipulator level2".S1 AND "PartHolderData".OKholderReadySideA AND NOT "PartHolderData".OKholderReadySideB;
      IF #_w1 AND ("PartHolderData".OkLowerStockAmountSideA = 0) THEN
          #prgNrForManipulatorDropoff := #jobManipulatorDropoff4;
      END_IF;
      IF #_w1 AND ("PartHolderData".OkLowerStockAmountSideA = 1) THEN
          #prgNrForManipulatorDropoff := #jobManipulatorDropoff5;
      END_IF;
      IF #_w1 AND ("PartHolderData".OkLowerStockAmountSideA = 2) THEN
          #prgNrForManipulatorDropoff := #jobManipulatorDropoff6;
      END_IF;
      #_w2 := #"Dropoff part to manipulator level2".S1 AND NOT "PartHolderData".OKholderReadySideA AND "PartHolderData".OKholderReadySideB;
      IF #_w2 AND ("PartHolderData".OkLowerStockAmountSideB = 0) THEN
          #prgNrForManipulatorDropoff := #jobManipulatorDropoff4;
      END_IF;
      IF #_w2 AND ("PartHolderData".OkLowerStockAmountSideB = 1) THEN
          #prgNrForManipulatorDropoff := #jobManipulatorDropoff5;
      END_IF;
      IF #_w2 AND ("PartHolderData".OkLowerStockAmountSideB = 2) THEN
          #prgNrForManipulatorDropoff := #jobManipulatorDropoff6;
      END_IF;
   NETWORK 3
      #base := "RobotMain_DB".RobotInStartingPosition AND "iR1ext";
   NETWORK 4
   TITLE = job start init
      "DevicesData".R1.Job.Start := FALSE;
   NETWORK 5
      "qR1_ST3free" := "sq_fitting_station_st3".base;

   // sequencer 1
   INITIAL_STEP Init:   // S1, max time T#10S, warning time T#7S
   END_STEP
   TRANSITION Trans1 FROM Init TO "Checking robot status"   // T1
      := ("ModeSelection_DB".mode.activeMode = "mode_2_base") OR (("ModeSelection_DB".mode.activeMode = "mode_4_semiautomat") AND #start);
   END_TRANSITION
   STEP Done:   // S2, max time T#10S, warning time T#7S
              N    "READER_MODEL_ACTUAL".ST2_CLEAR
   END_STEP
   TRANSITION Trans2 FROM Done TO "Wait for work for robot"   // T2, jump
      := TRUE;
   END_TRANSITION
   STEP "Base done":   // S12, max time T#10S, warning time T#7S
   END_STEP
   TRANSITION Trans17 FROM "Base done" TO "Wait for work for robot"   // T17
      := (("ModeSelection_DB".mode.activeMode = "mode_3_automat") OR (("ModeSelection_DB".mode.activeMode = "mode_4_semiautomat") AND #start)) AND (#"Base done".T > t#2000MS);
   END_TRANSITION
   STEP "Robot is not in starting position - move it to home manualy":   // S13, max time T#1S, warning time T#7S
      supervision V := #"Robot is not in starting position - move it to home manualy".T > #"Robot is not in starting position - move it to home manualy".T_MAX;
   END_STEP
   TRANSITION Trans18 FROM "Robot is not in starting position - move it to home manualy" TO "Base done"   // T18
      := "RobotMain_DB".RobotInStartingPosition;
   END_TRANSITION
   STEP "Robot in EXT?":   // S14, max time T#10S, warning time T#7S
      supervision V := #"Robot in EXT?".T > #"Robot in EXT?".T_MAX;
   END_STEP
   TRANSITION Trans19 FROM "Robot in EXT?" TO "Robot is not in starting position - move it to home manualy"   // T19
      := "iR1ext";
   END_TRANSITION
   STEP "Wait for work for robot":   // S15, max time T#10S, warning time T#7S
   END_STEP
   TRANSITION "jig dropoff" FROM "Wait for work for robot" TO "Dropoff part to jig"   // T22
      := (("ModeSelection_DB".mode.activeMode = "mode_3_automat") OR (("ModeSelection_DB".mode.activeMode = "mode_4_semiautomat") AND #start)) AND "RobotMain_DB".RobotInStartingPosition AND "sq_fitting_station_st3"."Waiting for the part to be inserted".X AND "DevicesData"."TA1-3MA".data.zones.outOfST3zone AND NOT "AutoPositions".St3_Fitting.PartPresent AND NOT "i3partPresent" AND "AutoPositions".R1_Gripper.PartPresent AND "iR1tubePresentFront" AND "iR1tubePresentRear" AND NOT "AutoPositions".R1_Gripper.StFinished[3] AND NOT "AutoPositions".R1_Gripper.PartNOK AND "sq_fitting_station_st3".base;
   END_TRANSITION
   TRANSITION "autoeject pickup" FROM "Wait for work for robot" TO "Pickup part from autoeject"   // T23
      := (("ModeSelection_DB".mode.activeMode = "mode_3_automat") OR (("ModeSelection_DB".mode.activeMode = "mode_4_semiautomat") AND #start)) AND "RobotMain_DB".RobotInStartingPosition AND "DevicesData"."TA1-3MA".data.zones.outOfOKposZone AND ((NOT "AutoInfo".EndProduction AND "AutoPositions".St3_Fitting.PartPresent) OR "AutoInfo".EndProduction) AND ("i4partPresent" OR "StationParameters".GhostMode) AND NOT "AutoPositions".R1_Gripper.PartPresent AND NOT "iR1tubePresentFront" AND NOT "iR1tubePresentRear" AND "AutoPositions".St4_OKposition.PartPresent;
   END_TRANSITION
   TRANSITION "manipulator dropoff" FROM "Wait for work for robot" TO "Which level?"   // T25
      := (("ModeSelection_DB".mode.activeMode = "mode_3_automat") OR (("ModeSelection_DB".mode.activeMode = "mode_4_semiautomat") AND #start)) AND "RobotMain_DB".RobotInStartingPosition AND (("PartHolderData".OKholderReadySideA AND (("PartHolderData".OkLowerStockAmountSideA < "StationParameters".OKLowerStockSize) OR ("PartHolderData".OkUpperStockAmountSideA < "StationParameters".OKUpperStockSize))) OR ("PartHolderData".OKholderReadySideB AND (("PartHolderData".OkLowerStockAmountSideB < "StationParameters".OKLowerStockSize) OR ("PartHolderData".OkUpperStockAmountSideB < "StationParameters".OKUpperStockSize)))) AND "AutoPositions".R1_Gripper.PartPresent AND "iR1tubePresentFront" AND "iR1tubePresentRear" AND "AutoPositions".R1_Gripper.StFinished[3] AND NOT "AutoPositions".R1_Gripper.PartNOK;
   END_TRANSITION
   TRANSITION "Mastering / brake test" FROM "Wait for work for robot" TO "Mastering?"   // T39
      := (("ModeSelection_DB".mode.activeMode = "mode_3_automat") OR (("ModeSelection_DB".mode.activeMode = "mode_4_semiautomat") AND #start)) AND "RobotMain_DB".RobotInStartingPosition AND "DevicesData"."TA1-3MA".data.zones.outOfST3zone AND NOT "AutoPositions".R1_Gripper.PartPresent AND NOT "iR1tubePresentFront" AND NOT "iR1tubePresentRear" AND ("AutoInfo".R1MasteringRequired OR "AutoInfo".R1BrakeTestRequired);
   END_TRANSITION
   TRANSITION "carousel pickup" FROM "Wait for work for robot" TO "Pickup part from carousel"   // T21
      := (("ModeSelection_DB".mode.activeMode = "mode_3_automat") OR (("ModeSelection_DB".mode.activeMode = "mode_4_semiautomat") AND #start)) AND "RobotMain_DB".RobotInStartingPosition AND "sq_carousel_unloading_st2"."Wait for robot to remove part".X AND "AutoPositions".St2_Table2.PartPresent AND (NOT "AutoPositions".St3_Fitting.PartPresent OR NOT "AutoPositions".St4_OKposition.PartPresent) AND NOT "AutoPositions".St2_Table2.PartNOK AND NOT "AutoPositions".R1_Gripper.PartPresent AND NOT "iR1tubePresentFront" AND NOT "iR1tubePresentRear" AND "iTableInPosition" AND "iTurnTableIndexerInPosition";
   END_TRANSITION
   TRANSITION home FROM "Wait for work for robot" TO "To home position"   // T38
      := (("ModeSelection_DB".mode.activeMode = "mode_3_automat") OR (("ModeSelection_DB".mode.activeMode = "mode_4_semiautomat") AND #start)) AND "iR1inPickupStartPositionAutoeject" AND "AutoInfo".EndProduction AND NOT "AutoPositions".St2_Table2.PartPresent AND "AutoPositions".St3_Fitting.PartPresent AND "i3partPresent" AND NOT "AutoPositions".St4_OKposition.PartPresent AND NOT "i4partPresent";
   END_TRANSITION
   STEP "Mastering job":   // S26, max time T#50S, warning time T#7S
      supervision V := #"Mastering job".T > #"Mastering job".T_MAX;
              N    "DevicesData".R1.Job.JobNr:=#jobMastering
              S    "DevicesData".R1.Job.Start
              R    "AutoInfo".R1MasteringRequired
   END_STEP
   TRANSITION Trans39 FROM "Mastering job" TO "Reset mastering request"   // T40
      := "DevicesData".R1.Job.Done;
   END_TRANSITION
   STEP "Dropoff part to jig":   // S19, max time T#30S, warning time T#7S
      supervision V := #"Dropoff part to jig".T > #"Dropoff part to jig".T_MAX;
              N    "DevicesData".R1.Job.JobNr:=#jobJigDropoff
              S    "DevicesData".R1.Job.Start
   END_STEP
   TRANSITION Trans31 FROM "Dropoff part to jig" TO Step32   // T31
      := "DevicesData".R1.Job.Done;
   END_TRANSITION
   STEP "Pickup part from autoeject":   // S20, max time T#30S, warning time T#7S
      supervision V := #"Pickup part from autoeject".T > #"Pickup part from autoeject".T_MAX;
              N    "DevicesData".R1.Job.JobNr:=#jobAutoEjectPickup
              S    "DevicesData".R1.Job.Start
   END_STEP
   TRANSITION Trans32 FROM "Pickup part from autoeject" TO Done   // T32
      := "DevicesData".R1.Job.Done;
   END_TRANSITION
   STEP "Which level?":   // S21, max time T#10S, warning time T#7S
   END_STEP
   TRANSITION top FROM "Which level?" TO "Dropoff part to manipulator level1"   // T33
      := (("PartHolderData".OKholderReadySideA AND ("PartHolderData".OkUpperStockAmountSideA < "StationParameters".OKUpperStockSize)) OR ("PartHolderData".OKholderReadySideB AND ("PartHolderData".OkUpperStockAmountSideB < "StationParameters".OKUpperStockSize))) AND NOT "StationParameters".DontUseHangerForParts;
   END_TRANSITION
   TRANSITION bottom FROM "Which level?" TO "Dropoff part to manipulator level2"   // T34
      := (("PartHolderData".OKholderReadySideA AND ("PartHolderData".OkLowerStockAmountSideA < "StationParameters".OKLowerStockSize)) OR ("PartHolderData".OKholderReadySideB AND ("PartHolderData".OkLowerStockAmountSideB < "StationParameters".OKLowerStockSize))) AND NOT "StationParameters".DontUseHangerForParts;
   END_TRANSITION
   TRANSITION "test only" FROM "Which level?" TO "Dropoff part to slide"   // T56
      := "StationParameters".DontUseHangerForParts;
   END_TRANSITION
   STEP "Dropoff part to manipulator level1":   // S22, max time T#30S, warning time T#7S
      supervision V := (#"Dropoff part to manipulator level1".T > #"Dropoff part to manipulator level1".T_MAX) AND (#"Dropoff part to manipulator level1".T > T#60S);
              N    "DevicesData".R1.Job.JobNr:=#prgNrForManipulatorDropoff
              S    "DevicesData".R1.Job.Start
   END_STEP
   TRANSITION Trans35 FROM "Dropoff part to manipulator level1" TO Done   // T35
      := "DevicesData".R1.Job.Done;
   END_TRANSITION
   STEP "Dropoff part to manipulator level2":   // S23, max time T#30S, warning time T#7S
      supervision V := #"Dropoff part to manipulator level2".T > #"Dropoff part to manipulator level2".T_MAX;
              N    "DevicesData".R1.Job.JobNr:=#prgNrForManipulatorDropoff
              S    "DevicesData".R1.Job.Start
   END_STEP
   TRANSITION Trans36 FROM "Dropoff part to manipulator level2" TO Done   // T36
      := "DevicesData".R1.Job.Done;
   END_TRANSITION
   STEP "Mastering?":   // S3, max time T#10S, warning time T#7S
   END_STEP
   TRANSITION Trans3 FROM "Mastering?" TO "Mastering required - press button to start"   // T3
      := NOT #startMastering AND NOT #startBraketest AND "AutoInfo".R1MasteringRequired;
   END_TRANSITION
   TRANSITION Trans42 FROM "Mastering?" TO "Braketest?"   // T42
      := NOT #startMastering AND NOT #startBraketest AND NOT "AutoInfo".R1MasteringRequired;
   END_TRANSITION
   STEP "Pickup part from carousel":   // S18, max time T#30S, warning time T#7S
      supervision V := #"Pickup part from carousel".T > #"Pickup part from carousel".T_MAX;
              N    "DevicesData".R1.Job.JobNr:=#jobCarouselPickup
              S    "DevicesData".R1.Job.Start
   END_STEP
   TRANSITION Trans30 FROM "Pickup part from carousel" TO Done   // T30
      := "DevicesData".R1.Job.Done;
   END_TRANSITION
   STEP "Braketest?":   // S27, max time T#10S, warning time T#7S
   END_STEP
   TRANSITION Trans41 FROM "Braketest?" TO "Braketest required - press button to start"   // T41
      := "AutoInfo".R1BrakeTestRequired;
   END_TRANSITION
   TRANSITION Trans44 FROM "Braketest?" TO Done   // T44
      := NOT "AutoInfo".R1BrakeTestRequired;
   END_TRANSITION
   STEP "BrakeCheck job":   // S28, max time T#60S, warning time T#7S
      supervision V := #"BrakeCheck job".T > #"BrakeCheck job".T_MAX;
              N    "DevicesData".R1.Job.JobNr:=#jobBreaktest
              S    "DevicesData".R1.Job.Start
              R    "AutoInfo".R1BrakeTestRequired
   END_STEP
   TRANSITION Trans40 FROM "BrakeCheck job" TO "Reset braketest request"   // T43
      := "DevicesData".R1.Job.Done;
   END_TRANSITION
   STEP "Reset mastering request":   // S29, max time T#10S, warning time T#7S
              R    "AutoInfo".R1MasteringRequired
   END_STEP
   TRANSITION Trans45 FROM "Reset mastering request" TO "Braketest?"   // T45
      := TRUE;
   END_TRANSITION
   STEP "Reset braketest request":   // S30, max time T#10S, warning time T#7S
              R    "AutoInfo".R1BrakeTestRequired
   END_STEP
   TRANSITION Trans46 FROM "Reset braketest request" TO Done   // T46
      := TRUE;
   END_TRANSITION
   STEP "Mastering required - press button to start":   // S34, max time T#10S, warning time T#7S
   END_STEP
   TRANSITION Trans53 FROM "Mastering required - press button to start" TO "Mastering job"   // T53
      := #startMastering;
   END_TRANSITION
   STEP "Braketest required - press button to start":   // S35, max time T#10S, warning time T#7S
   END_STEP
   TRANSITION Trans54 FROM "Braketest required - press button to start" TO "BrakeCheck job"   // T54
      := #startBraketest;
   END_TRANSITION
   STEP "Checking robot status":   // S36, max time T#10S, warning time T#7S
   END_STEP
   TRANSITION Trans55 FROM "Checking robot status" TO "Robot in EXT?"   // T55
      := "iR1pgNoReq";
   END_TRANSITION
   STEP "Dropoff part to slide":   // S24, max time T#40S, warning time T#7S
      supervision V := #"Dropoff part to slide".T > #"Dropoff part to slide".T_MAX;
              N    "DevicesData".R1.Job.JobNr:=#jobManipulatorForTesting
              S    "DevicesData".R1.Job.Start
   END_STEP
   TRANSITION Trans37 FROM "Dropoff part to slide" TO Done   // T37
      := "DevicesData".R1.Job.Done;
   END_TRANSITION
   STEP "To home position":   // S25, max time T#10S, warning time T#7S
      supervision V := #"To home position".T > #"To home position".T_MAX;
              N    "DevicesData".R1.Job.JobNr:=#jobHoming
              S    "DevicesData".R1.Job.Start
   END_STEP
   TRANSITION Trans33 FROM "To home position" TO Done   // T47
      := "DevicesData".R1.Job.Done;
   END_TRANSITION
   STEP Step32:   // S32, max time T#10S, warning time T#7S
   END_STEP
   TRANSITION Trans49 FROM Step32 TO Done   // T49
      := TRUE;
   END_TRANSITION

   // permanent post-instructions
   NETWORK 1
      IF #startMastering THEN #startMastering := FALSE; END_IF;
      IF #startBraketest THEN #startBraketest := FALSE; END_IF;
END_FUNCTION_BLOCK

FUNCTION "Reader Cognex Dataman" : Void   // FC302, LAD
{ S7_Optimized_Access := 'TRUE' }
VERSION : 0.1
// stored: AutoNumber false, IsIECCheckEnabled false, SetENOAutomatically false, UDAEnableTagReadback false
   VAR_IN_OUT
      ID : "UDT_CognexReaders";
   END_VAR
   VAR_TEMP
      AcquisitionControl : Struct
         TriggerEnable : Bool;
         Trigger : Bool;
         Reserved : Array[2..7] of Bool;
      END_STRUCT;
      AcquisitionStatus : Struct
         TriggerReady : Bool;
         TriggerAck : Bool;
         Reserved : Bool;
         MissedAck : Bool;
         Reserved_1 : Array[4..7] of Bool;
         TriggerID : Word;
      END_STRUCT;
      ResultsControl : Struct
         ResultBufferEnable : Bool;
         ResultsAck : Bool;
         Reserve : Array[2..7] of Bool;
      END_STRUCT;
      ResultsStatus : Struct
         Decoding : Bool;
         "Decode Complete" : Bool;
         "Results Buffer Overrun" : Bool;
         "Results Available" : Bool;
         Reserve_4 : Bool;
         Reserve_5 : Bool;
         Reserve_6 : Bool;
         GeneralFault : Bool;
      END_STRUCT;
      ResultData : Struct
         ID : Word;
         Code : Word;
         Lenght : Word;
         Data : Array[1..64] of Byte;
      END_STRUCT;
      "Return" : Word;
   END_VAR
   VAR_TEMP   // added for the SCL form of the ladder/FBD networks
      _w1 : Bool;
   END_VAR
BEGIN

REGION Network 1: Read input map
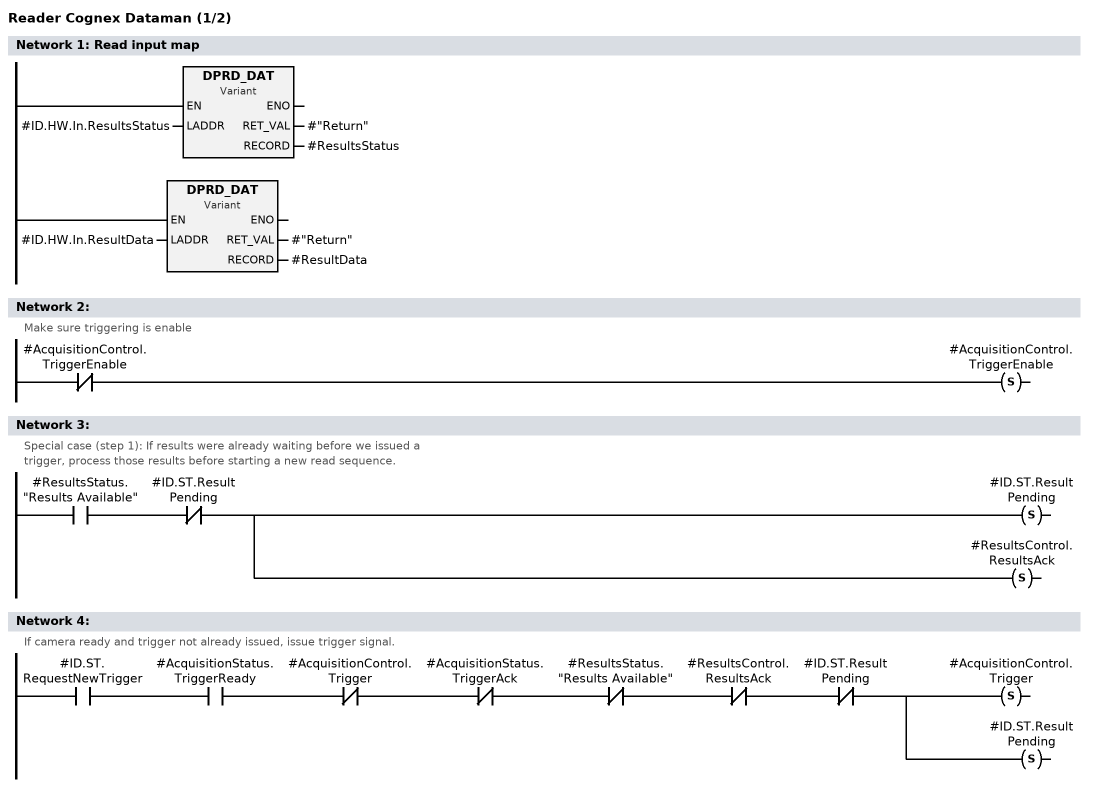
   RUNG wire#powerrail
      { S7_Templates := "[ptr_type := Variant, laddr_type := HW_IO]" } DPRD_DAT(LADDR := #ID.HW.In.ResultsStatus, RET_VAL => #"Return", RECORD => #ResultsStatus)
   END_RUNG
   RUNG wire#powerrail
      { S7_Templates := "[ptr_type := Variant, laddr_type := HW_IO]" } DPRD_DAT(LADDR := #ID.HW.In.ResultData, RET_VAL => #"Return", RECORD => #ResultData)
   END_RUNG
   // the same network as SCL:
   #"Return" := DPRD_DAT(LADDR := #ID.HW.In.ResultsStatus, RECORD => #ResultsStatus);
   #"Return" := DPRD_DAT(LADDR := #ID.HW.In.ResultData, RECORD => #ResultData);
END_REGION

REGION Network 2
   // Make sure triggering is enable
   RUNG wire#powerrail
      I_Contact( #AcquisitionControl.TriggerEnable )
      S_Coil( #AcquisitionControl.TriggerEnable )
   END_RUNG
   // the same network as SCL:
   IF NOT #AcquisitionControl.TriggerEnable THEN #AcquisitionControl.TriggerEnable := TRUE; END_IF;
END_REGION

REGION Network 3
   // Special case (step 1): If results were already waiting before we issued a 
   // trigger, process those results before starting a new read sequence.
   RUNG wire#powerrail
      Contact( #ResultsStatus."Results Available" )
      I_Contact( #ID.ST.ResultPending )
      wire#w1
      S_Coil( #ID.ST.ResultPending )
   END_RUNG
   RUNG wire#w1
      S_Coil( #ResultsControl.ResultsAck )
   END_RUNG
   // the same network as SCL:
   #_w1 := #ResultsStatus."Results Available" AND NOT #ID.ST.ResultPending;
   IF #_w1 THEN
       #ID.ST.ResultPending := TRUE;
       #ResultsControl.ResultsAck := TRUE;
   END_IF;
END_REGION

REGION Network 4
   // If camera ready and trigger not already issued, issue trigger signal.
   RUNG wire#powerrail
      Contact( #ID.ST.RequestNewTrigger )
      Contact( #AcquisitionStatus.TriggerReady )
      I_Contact( #AcquisitionControl.Trigger )
      I_Contact( #AcquisitionStatus.TriggerAck )
      I_Contact( #ResultsStatus."Results Available" )
      I_Contact( #ResultsControl.ResultsAck )
      I_Contact( #ID.ST.ResultPending )
      wire#w1
      S_Coil( #AcquisitionControl.Trigger )
   END_RUNG
   RUNG wire#w1
      S_Coil( #ID.ST.ResultPending )
   END_RUNG
   // the same network as SCL:
   #_w1 := #ID.ST.RequestNewTrigger AND #AcquisitionStatus.TriggerReady AND NOT #AcquisitionControl.Trigger AND NOT #AcquisitionStatus.TriggerAck AND NOT #ResultsStatus."Results Available" AND NOT #ResultsControl.ResultsAck AND NOT #ID.ST.ResultPending;
   IF #_w1 THEN
       #AcquisitionControl.Trigger := TRUE;
       #ID.ST.ResultPending := TRUE;
   END_IF;
END_REGION

